//     Task_P2Main Outputs/GMotion.arrAxis[166].PlcToNc <-> Inputs/FromPlc
//   DPPLC/DPPLC Instance <-> NC-Task 1 SAF/Axes/Axis194_167 P3_M2_OvenRetracting
//     Task_P2Main Inputs/GMotion.arrAxis[167].NcToPlc <-> Outputs/ToPlc
//     Task_P2Main Outputs/GMotion.arrAxis[167].PlcToNc <-> Inputs/FromPlc
//   DPPLC/DPPLC Instance <-> NC-Task 1 SAF/Axes/Axis195_168 P3_M2_OvenUpDown
//     Task_P2Main Inputs/GMotion.arrAxis[168].NcToPlc <-> Outputs/ToPlc
//     Task_P2Main Outputs/GMotion.arrAxis[168].PlcToNc <-> Inputs/FromPlc
//   DPPLC/DPPLC Instance <-> NC-Task 1 SAF/Axes/Axis196_169 P3_M3_HotPressingLine
//     Task_P2Main Inputs/GMotion.arrAxis[169].NcToPlc <-> Outputs/ToPlc
//     Task_P2Main Outputs/GMotion.arrAxis[169].PlcToNc <-> Inputs/FromPlc
//   DPPLC/DPPLC Instance <-> NC-Task 1 SAF/Axes/Axis197_170 P3_M3_HotPressingActuated
//     Task_P2Main Inputs/GMotion.arrAxis[170].NcToPlc <-> Outputs/ToPlc
//     Task_P2Main Outputs/GMotion.arrAxis[170].PlcToNc <-> Inputs/FromPlc
//   DPPLC/DPPLC Instance <-> NC-Task 1 SAF/Axes/Axis198_171  P3_M4_WeighLine
//     Task_P2Main Inputs/GMotion.arrAxis[171].NcToPlc <-> Outputs/ToPlc
//     Task_P2Main Outputs/GMotion.arrAxis[171].PlcToNc <-> Inputs/FromPlc
//   DPPLC/DPPLC Instance <-> NC-Task 1 SAF/Axes/Axis199_172 P3_M4_WeighUpDown
//     Task_P2Main Inputs/GMotion.arrAxis[172].NcToPlc <-> Outputs/ToPlc
//     Task_P2Main Outputs/GMotion.arrAxis[172].PlcToNc <-> Inputs/FromPlc
//   DPPLC/DPPLC Instance <-> NC-Task 1 SAF/Axes/Axis200_173 P3_M4_WeighWhirling
//     Task_P2Main Inputs/GMotion.arrAxis[173].NcToPlc <-> Outputs/ToPlc
//     Task_P2Main Outputs/GMotion.arrAxis[173].PlcToNc <-> Inputs/FromPlc
//   DPPLC/DPPLC Instance <-> NC-Task 1 SAF/Axes/Axis201_174 P3_M4_SortingoutCarrying
//     Task_P2Main Inputs/GMotion.arrAxis[174].NcToPlc <-> Outputs/ToPlc
//     Task_P2Main Outputs/GMotion.arrAxis[174].PlcToNc <-> Inputs/FromPlc
//   DPPLC/DPPLC Instance <-> NC-Task 1 SAF/Axes/Axis202_175 P3_M4_SortingoutUpDown
//     Task_P2Main Inputs/GMotion.arrAxis[175].NcToPlc <-> Outputs/ToPlc
//     Task_P2Main Outputs/GMotion.arrAxis[175].PlcToNc <-> Inputs/FromPlc
//   DPPLC/DPPLC Instance <-> NC-Task 1 SAF/Axes/Axis203_176 P3_M4_OffloadingCarrying
//     Task_P2Main Inputs/GMotion.arrAxis[176].NcToPlc <-> Outputs/ToPlc
//     Task_P2Main Outputs/GMotion.arrAxis[176].PlcToNc <-> Inputs/FromPlc
//   DPPLC/DPPLC Instance <-> NC-Task 1 SAF/Axes/Axis204_177 P3_M4_OffloadingUpDown
//     Task_P2Main Inputs/GMotion.arrAxis[177].NcToPlc <-> Outputs/ToPlc
//     Task_P2Main Outputs/GMotion.arrAxis[177].PlcToNc <-> Inputs/FromPlc
//   DPPLC/DPPLC Instance <-> NC-Task 1 SAF/Axes/Axis205_178 P3_TapeAdvance
//     Task_P2Main Inputs/GMotion.arrAxis[178].NcToPlc <-> Outputs/ToPlc
//     Task_P2Main Outputs/GMotion.arrAxis[178].PlcToNc <-> Inputs/FromPlc
//   DPPLC/DPPLC Instance <-> NC-Task 1 SAF/Axes/Axis206_179 P3_TapeTranslation
//     Task_P2Main Inputs/GMotion.arrAxis[179].NcToPlc <-> Outputs/ToPlc
//     Task_P2Main Outputs/GMotion.arrAxis[179].PlcToNc <-> Inputs/FromPlc
//   DPPLC/DPPLC Instance <-> NC-Task 1 SAF/Axes/Axis207_180 P3_IDPut
//     Task_P2Main Inputs/GMotion.arrAxis[180].NcToPlc <-> Outputs/ToPlc
//     Task_P2Main Outputs/GMotion.arrAxis[180].PlcToNc <-> Inputs/FromPlc
//   DPPLC/DPPLC Instance <-> NC-Task 1 SAF/Axes/Axis208_181 P3_IDLift
//     Task_P2Main Inputs/GMotion.arrAxis[181].NcToPlc <-> Outputs/ToPlc
//     Task_P2Main Outputs/GMotion.arrAxis[181].PlcToNc <-> Inputs/FromPlc
//   DPPLC/DPPLC Instance <-> NC-Task 1 SAF/Axes/Axis209_182 P3_Standby5
//     Task_P2Main Inputs/GMotion.arrAxis[182].NcToPlc <-> Outputs/ToPlc
//     Task_P2Main Outputs/GMotion.arrAxis[182].PlcToNc <-> Inputs/FromPlc
//   DPPLC/DPPLC Instance <-> NC-Task 1 SAF/Axes/Axis218_153 P2M2_VirTimeWind
//     Task_P2Main Inputs/GMotion.arrAxis[153].NcToPlc <-> Outputs/ToPlc
//     Task_P2Main Outputs/GMotion.arrAxis[153].PlcToNc <-> Inputs/FromPlc
//   DPPLC/DPPLC Instance <-> NC-Task 1 SAF/Axes/Axis219_154 P2M3_VirTimeWind
//     Task_P2Main Inputs/GMotion.arrAxis[154].NcToPlc <-> Outputs/ToPlc
//     Task_P2Main Outputs/GMotion.arrAxis[154].PlcToNc <-> Inputs/FromPlc
//   DPPLC/DPPLC Instance <-> NC-Task 1 SAF/Axes/Axis220_140 P2M1_VirTimeWind
//     Task_P2Main Inputs/GMotion.arrAxis[140].NcToPlc <-> Outputs/ToPlc
//     Task_P2Main Outputs/GMotion.arrAxis[140].PlcToNc <-> Inputs/FromPlc
//   DPPLC/DPPLC Instance <-> NC-Task 1 SAF/Axes/Axis221_141 P2M1_VirMain
//     Task_P2Main Inputs/GMotion.arrAxis[141].NcToPlc <-> Outputs/ToPlc
//     Task_P2Main Outputs/GMotion.arrAxis[141].PlcToNc <-> Inputs/FromPlc
//   DPPLC/DPPLC Instance <-> NC-Task 1 SAF/Axes/Axis222_142 P2M1_VirDriver
//     Task_P2Main Inputs/GMotion.arrAxis[142].NcToPlc <-> Outputs/ToPlc
//     Task_P2Main Outputs/GMotion.arrAxis[142].PlcToNc <-> Inputs/FromPlc
//   DPPLC/DPPLC Instance <-> NC-Task 1 SAF/Axes/Axis223_143 P2M1_VirTailCurl
//     Task_P2Main Inputs/GMotion.arrAxis[143].NcToPlc <-> Outputs/ToPlc
//     Task_P2Main Outputs/GMotion.arrAxis[143].PlcToNc <-> Inputs/FromPlc
//   DPPLC/DPPLC Instance <-> NC-Task 1 SAF/Axes/Axis224_144  P2M1VirGM
//     Task_P2Main Inputs/GMotion.arrAxis[144].NcToPlc <-> Outputs/ToPlc
//     Task_P2Main Outputs/GMotion.arrAxis[144].PlcToNc <-> Inputs/FromPlc
//   DPPLC/DPPLC Instance <-> NC-Task 1 SAF/Axes/Axis225_145 P2M2_VirMain
//     Task_P2Main Inputs/GMotion.arrAxis[145].NcToPlc <-> Outputs/ToPlc
//     Task_P2Main Outputs/GMotion.arrAxis[145].PlcToNc <-> Inputs/FromPlc
//   DPPLC/DPPLC Instance <-> NC-Task 1 SAF/Axes/Axis226_146 P2M2_VirDriver
//     Task_P2Main Inputs/GMotion.arrAxis[146].NcToPlc <-> Outputs/ToPlc
//     Task_P2Main Outputs/GMotion.arrAxis[146].PlcToNc <-> Inputs/FromPlc
//   DPPLC/DPPLC Instance <-> NC-Task 1 SAF/Axes/Axis227_147 P2M2_VirTailCurl
//     Task_P2Main Inputs/GMotion.arrAxis[147].NcToPlc <-> Outputs/ToPlc
//     Task_P2Main Outputs/GMotion.arrAxis[147].PlcToNc <-> Inputs/FromPlc
//   DPPLC/DPPLC Instance <-> NC-Task 1 SAF/Axes/Axis228_148  P2M2VirGM
//     Task_P2Main Inputs/GMotion.arrAxis[148].NcToPlc <-> Outputs/ToPlc
//     Task_P2Main Outputs/GMotion.arrAxis[148].PlcToNc <-> Inputs/FromPlc
//   DPPLC/DPPLC Instance <-> NC-Task 1 SAF/Axes/Axis229_149 P2M3_VirMain
//     Task_P2Main Inputs/GMotion.arrAxis[149].NcToPlc <-> Outputs/ToPlc
//     Task_P2Main Outputs/GMotion.arrAxis[149].PlcToNc <-> Inputs/FromPlc
//   DPPLC/DPPLC Instance <-> NC-Task 1 SAF/Axes/Axis230_150 P2M3_VirDriver
//     Task_P2Main Inputs/GMotion.arrAxis[150].NcToPlc <-> Outputs/ToPlc
//     Task_P2Main Outputs/GMotion.arrAxis[150].PlcToNc <-> Inputs/FromPlc
//   DPPLC/DPPLC Instance <-> NC-Task 1 SAF/Axes/Axis231_151 P2M3_VirTailCurl
//     Task_P2Main Inputs/GMotion.arrAxis[151].NcToPlc <-> Outputs/ToPlc
//     Task_P2Main Outputs/GMotion.arrAxis[151].PlcToNc <-> Inputs/FromPlc
//   DPPLC/DPPLC Instance <-> NC-Task 1 SAF/Axes/Axis232  P2M3VirGM
//     Task_P2Main Inputs/GMotion.arrAxis[152].NcToPlc <-> Outputs/ToPlc
//     Task_P2Main Outputs/GMotion.arrAxis[152].PlcToNc <-> Inputs/FromPlc
//   DPPLC/DPPLC Instance <-> MQPLC/MQPLC Instance
//     Task_P2M3 Inputs/IO.M_Pro <-> Task_P1 Outputs/IO.M_Pro
//     Task_P2M3 Outputs/IO.D_Pro <-> Task_P1 Inputs/IO.D_Pro
//     Task_P2M3 Outputs/IO.D_Sys/P3ReadParDone <-> Task_P1 Inputs/IO.D_Sys/P3ReadParDone
//     Task_P2M3 Outputs/IO.D_Sys/P3SaveParDone <-> Task_P1 Inputs/IO.D_Sys/P3SaveParDone
//     Task_P2M3 Outputs/IO.D_Sys/bP2ClearDo <-> Task_P1 Inputs/IO.D_Sys/bP2ClearDo
//     Task_P2M3 Outputs/IO.D_Sys/bP2ClearDone <-> Task_P1 Inputs/IO.D_Sys/bP2ClearDone
//     Task_P2M3 Outputs/IO.D_Sys/bP2Estop <-> Task_P1 Inputs/IO.D_Sys/bP2Estop
//     Task_P2M3 Outputs/IO.D_Sys/bP2M1Enable <-> Task_P1 Inputs/IO.D_Sys/bP2M1Enable
//     Task_P2M3 Outputs/IO.D_Sys/bP2M2Enable <-> Task_P1 Inputs/IO.D_Sys/bP2M2Enable
//     Task_P2M3 Outputs/IO.D_Sys/bP2M3Enable <-> Task_P1 Inputs/IO.D_Sys/bP2M3Enable
//     Task_P2M3 Outputs/IO.D_Sys/bP2Runing <-> Task_P1 Inputs/IO.D_Sys/bP2Runing
//     Task_P2M3 Outputs/IO.D_Sys/bP2Start <-> Task_P1 Inputs/IO.D_Sys/bP2Start
//     Task_P2M3 Outputs/IO.D_Sys/fM1MainSetPos <-> Task_P1 Inputs/IO.D_Sys/fM1MainSetPos
//     Task_P2M3 Outputs/IO.D_Sys/fM2MainSetPos <-> Task_P1 Inputs/IO.D_Sys/fM2MainSetPos
//     Task_P2M3 Outputs/IO.D_Sys/fM3MainSetPos <-> Task_P1 Inputs/IO.D_Sys/fM3MainSetPos
//     Task_P2M3 Outputs/IO.D_Sys/iAn1Ask <-> Task_P1 Inputs/IO.D_Sys/iAn1Ask
//     Task_P2M3 Outputs/IO.D_Sys/iAn2Ask <-> Task_P1 Inputs/IO.D_Sys/iAn2Ask
//     Task_P2M3 Outputs/IO.D_Sys/iAn3Ask <-> Task_P1 Inputs/IO.D_Sys/iAn3Ask
//     Task_P2M3 Outputs/IO.D_Sys/iCa1Ask <-> Task_P1 Inputs/IO.D_Sys/iCa1Ask
//     Task_P2M3 Outputs/IO.D_Sys/iCa2Ask <-> Task_P1 Inputs/IO.D_Sys/iCa2Ask
//     Task_P2M3 Outputs/IO.D_Sys/iCa3Ask <-> Task_P1 Inputs/IO.D_Sys/iCa3Ask
//     Task_P2Main Inputs/IO.AnMQ_MES1 <-> Task_P1 Outputs/IO.AnMQ_MES1
//     Task_P2Main Inputs/IO.AnMQ_MES2 <-> Task_P1 Outputs/IO.AnMQ_MES2
//     Task_P2Main Inputs/IO.AnMQ_MES3 <-> Task_P1 Outputs/IO.AnMQ_MES3
//     Task_P2Main Inputs/IO.CaMQ_MES1 <-> Task_P1 Outputs/IO.CaMQ_MES1
//     Task_P2Main Inputs/IO.CaMQ_MES2 <-> Task_P1 Outputs/IO.CaMQ_MES2
//     Task_P2Main Inputs/IO.CaMQ_MES3 <-> Task_P1 Outputs/IO.CaMQ_MES3
//     Task_P2Main Outputs/IO.YL_Q <-> Task_P1 Inputs/IO.YL_I
//     Task_P3 Inputs/IO.M_Sys/P1ReadParDone <-> Task_P1 Outputs/IO.M_Sys/P1ReadParDone
//     Task_P3 Inputs/IO.M_Sys/P1SaveParDone <-> Task_P1 Outputs/IO.M_Sys/P1SaveParDone
//     Task_P3 Inputs/IO.M_Sys/bP1ClearDo <-> Task_P1 Outputs/IO.M_Sys/bP1ClearDo
//     Task_P3 Inputs/IO.M_Sys/bP1ClearDone <-> Task_P1 Outputs/IO.M_Sys/bP1ClearDone
//     Task_P3 Inputs/IO.M_Sys/bP1Estop <-> Task_P1 Outputs/IO.M_Sys/bP1Estop
//     Task_P3 Inputs/IO.M_Sys/bP1Runing <-> Task_P1 Outputs/IO.M_Sys/bP1Runing
//     Task_P3 Inputs/IO.M_Sys/bP1Start <-> Task_P1 Outputs/IO.M_Sys/bP1Start
//     Task_P3 Inputs/IO.M_Sys/iCarryPoleMode <-> Task_P1 Outputs/IO.M_Sys/iCarryPoleMode
//     Task_P3 Inputs/IO.M_Sys/p1state <-> Task_P1 Outputs/IO.M_Sys/p1state
//     Task_P3 Inputs/IO.YL_INT1 <-> Task_P1 Outputs/IO.YL_INT1
//     Task_P3 Inputs/P3IO.MTD_Mes1/bFuncEN <-> Task_P1 Outputs/IO.MTD_Mes1/bFuncEN
//     Task_P3 Inputs/P3IO.MTD_Mes1/rExcelRate <-> Task_P1 Outputs/IO.MTD_Mes1/rExcelRate
//     Task_P3 Inputs/P3IO.MTD_Mes1/uOther <-> Task_P1 Outputs/IO.MTD_Mes1/uOther
//     Task_P3 Inputs/P3Par.MQ_To_DT_MES <-> Task_P1 Outputs/IO.MQ_To_DT_MES
//     Task_P3 Outputs/IO.YL_INT2 <-> Task_P1 Inputs/IO.YL_INT2
//     Task_P3 Outputs/P3IO.DTM_Mes1/bFuncEN <-> Task_P1 Inputs/IO.DTM_Mes1/bFuncEN
//     Task_P3 Outputs/P3IO.DTM_Mes1/uOther <-> Task_P1 Inputs/IO.DTM_Mes1/uOther
//     Task_P3 Outputs/P3Par.DT_To_MQ_MES <-> Task_P1 Inputs/IO.DT_To_MQ_MES
//   MQPLC/MQPLC Instance <-> Device 3 (EtherCAT)/Box 2 (CU1128)/Term 24 (CU1128-B)/负极上表面除尘皮带(InoSV660N)
//     Task_P1 Inputs/GMotion.DrivesOP[42] <-> InfoData/State
//     Task_P1 Inputs/GMotion.arrAxisCtrl[42].Io.DigitalInputs <-> Inputs/Digital inputs
//     Task_P1 Inputs/GMotion.arrAxisCtrl[42].Io.ErrorCode <-> Inputs/Error code
//     Task_P1 Inputs/GMotion.iActTorque_M[42] <-> Inputs/Torque actual value
//   MQPLC/MQPLC Instance <-> Device 3 (EtherCAT)/Box 2 (CU1128)/Term 24 (CU1128-B)/负极下表面除尘倒装皮带(InoSV660N)
//     Task_P1 Inputs/GMotion.DrivesOP[43] <-> InfoData/State
//     Task_P1 Inputs/GMotion.arrAxisCtrl[43].Io.DigitalInputs <-> Inputs/Digital inputs
//     Task_P1 Inputs/GMotion.arrAxisCtrl[43].Io.ErrorCode <-> Inputs/Error code
//     Task_P1 Inputs/GMotion.iActTorque_M[43] <-> Inputs/Torque actual value
//   MQPLC/MQPLC Instance <-> Device 3 (EtherCAT)/Box 2 (CU1128)/Term 24 (CU1128-B)/负极倒角模具(InoSV660N)
//     Task_P1 Inputs/GMotion.DrivesOP[30] <-> InfoData/State
//     Task_P1 Inputs/GMotion.arrAxisCtrl[30].Io.DigitalInputs <-> Inputs/Digital inputs
//     Task_P1 Inputs/GMotion.arrAxisCtrl[30].Io.ErrorCode <-> Inputs/Error code
//     Task_P1 Inputs/GMotion.iActTorque_M[30] <-> Inputs/Torque actual value
//   MQPLC/MQPLC Instance <-> Device 3 (EtherCAT)/Box 2 (CU1128)/Term 24 (CU1128-B)/负极右放卷电机(InoSV660N)
//     Task_P1 Inputs/GMotion.DrivesOP[26] <-> InfoData/State
//     Task_P1 Inputs/GMotion.arrAxisCtrl[26].Io.DigitalInputs <-> Inputs/Digital inputs
//     Task_P1 Inputs/GMotion.arrAxisCtrl[26].Io.ErrorCode <-> Inputs/Error code
//     Task_P1 Inputs/GMotion.iActTorque_M[26] <-> Inputs/Torque actual value
//   MQPLC/MQPLC Instance <-> Device 3 (EtherCAT)/Box 2 (CU1128)/Term 24 (CU1128-B)/负极尺寸CCD压片升降(InoSV660N)
//     Task_P1 Inputs/GMotion.DrivesOP[38] <-> InfoData/State
//     Task_P1 Inputs/GMotion.arrAxisCtrl[38].Io.DigitalInputs <-> Inputs/Digital inputs
//     Task_P1 Inputs/GMotion.arrAxisCtrl[38].Io.ErrorCode <-> Inputs/Error code
//     Task_P1 Inputs/GMotion.iActTorque_M[38] <-> Inputs/Torque actual value
//   MQPLC/MQPLC Instance <-> Device 3 (EtherCAT)/Box 2 (CU1128)/Term 24 (CU1128-B)/负极左放卷电机(InoSV660N)
//     Task_P1 Inputs/GMotion.DrivesOP[25] <-> InfoData/State
//     Task_P1 Inputs/GMotion.arrAxisCtrl[25].Io.DigitalInputs <-> Inputs/Digital inputs
//     Task_P1 Inputs/GMotion.arrAxisCtrl[25].Io.ErrorCode <-> Inputs/Error code
//     Task_P1 Inputs/GMotion.iActTorque_M[25] <-> Inputs/Torque actual value
//   MQPLC/MQPLC Instance <-> Device 3 (EtherCAT)/Box 2 (CU1128)/Term 24 (CU1128-B)/负极模具纠偏X轴(肩宽)(InoSV660N)
//     Task_P1 Inputs/GMotion.DrivesOP[31] <-> InfoData/State
//     Task_P1 Inputs/GMotion.arrAxisCtrl[31].Io.DigitalInputs <-> Inputs/Digital inputs
//     Task_P1 Inputs/GMotion.arrAxisCtrl[31].Io.ErrorCode <-> Inputs/Error code
//     Task_P1 Inputs/GMotion.iActTorque_M[31] <-> Inputs/Torque actual value
//   MQPLC/MQPLC Instance <-> Device 3 (EtherCAT)/Box 2 (CU1128)/Term 24 (CU1128-B)/负极模具纠偏Y轴(InoSV660N)
//     Task_P1 Inputs/GMotion.DrivesOP[32] <-> InfoData/State
//     Task_P1 Inputs/GMotion.arrAxisCtrl[32].Io.DigitalInputs <-> Inputs/Digital inputs
//     Task_P1 Inputs/GMotion.arrAxisCtrl[32].Io.ErrorCode <-> Inputs/Error code
//     Task_P1 Inputs/GMotion.iActTorque_M[32] <-> Inputs/Torque actual value
//   MQPLC/MQPLC Instance <-> Device 3 (EtherCAT)/Box 2 (CU1128)/Term 24 (CU1128-B)/负极模切主驱动(CDHD)
//     Task_P1 Inputs/GMotion.DrivesOP[33] <-> InfoData/State
//     Task_P1 Inputs/GMotion.arrAxisCtrl[33].Io.DigitalInputs <-> TxPDO 4/Digital inputs
//     Task_P1 Inputs/GMotion.iActTorque_M[33] <-> TxPDO 1/Torque Actual Value
//   MQPLC/MQPLC Instance <-> Device 3 (EtherCAT)/Box 2 (CU1128)/Term 24 (CU1128-B)/负极模切前摆杆张力(InoSV660N)
//     Task_P1 Inputs/GMotion.DrivesOP[27] <-> InfoData/State
//     Task_P1 Inputs/GMotion.arrAxisCtrl[27].Io.DigitalInputs <-> Inputs/Digital inputs
//     Task_P1 Inputs/GMotion.arrAxisCtrl[27].Io.ErrorCode <-> Inputs/Error code
//     Task_P1 Inputs/GMotion.iActDriveTorque[2] <-> Inputs/Torque actual value
//     Task_P1 Outputs/GMotion.iMaxProfileVelo[2] <-> Outputs/Max profile velocity
//     Task_P1 Outputs/GMotion.iNegtiveTorqueLimits[2] <-> Outputs/Negative torque limit value
//     Task_P1 Outputs/GMotion.iPostiveTorqueLimits[2] <-> Outputs/Positive torque limit value
//     Task_P1 Outputs/GMotion.iSetDriveMode[2] <-> Outputs/Modes of operation
//     Task_P1 Outputs/GMotion.iTargetTorque[2] <-> Outputs/Target torque
//   MQPLC/MQPLC Instance <-> Device 3 (EtherCAT)/Box 2 (CU1128)/Term 24 (CU1128-B)/负极模切极片缓存(CDHD)
//     Task_P1 Inputs/GMotion.DrivesOP[29] <-> InfoData/State
//     Task_P1 Inputs/GMotion.arrAxisCtrl[29].Io.DigitalInputs <-> TxPDO 4/Digital inputs
//     Task_P1 Inputs/GMotion.iActTorque_M[29] <-> TxPDO 1/Torque Actual Value
//   MQPLC/MQPLC Instance <-> Device 3 (EtherCAT)/Box 2 (CU1128)/Term 24 (CU1128-B)/负极模切辅助驱动(InoSV660N)
//     Task_P1 Inputs/GMotion.DrivesOP[28] <-> InfoData/State
//     Task_P1 Inputs/GMotion.arrAxisCtrl[28].Io.DigitalInputs <-> Inputs/Digital inputs
//     Task_P1 Inputs/GMotion.arrAxisCtrl[28].Io.ErrorCode <-> Inputs/Error code
//     Task_P1 Inputs/GMotion.iActTorque_M[28] <-> Inputs/Torque actual value
//   MQPLC/MQPLC Instance <-> Device 3 (EtherCAT)/Box 2 (CU1128)/Term 24 (CU1128-B)/负极裁切切刀(InoSV660N)
//     Task_P1 Inputs/GMotion.DrivesOP[34] <-> InfoData/State
//     Task_P1 Inputs/GMotion.arrAxisCtrl[34].Io.DigitalInputs <-> Inputs/Digital inputs
//     Task_P1 Inputs/GMotion.arrAxisCtrl[34].Io.ErrorCode <-> Inputs/Error code
//     Task_P1 Inputs/GMotion.iActTorque_M[34] <-> Inputs/Torque actual value
//   MQPLC/MQPLC Instance <-> Device 3 (EtherCAT)/Box 2 (CU1128)/Term 24 (CU1128-B)/负极裁切角度纠偏(InoSV660N)
//     Task_P1 Inputs/GMotion.DrivesOP[35] <-> InfoData/State
//     Task_P1 Inputs/GMotion.arrAxisCtrl[35].Io.DigitalInputs <-> Inputs/Digital inputs
//     Task_P1 Inputs/GMotion.arrAxisCtrl[35].Io.ErrorCode <-> Inputs/Error code
//     Task_P1 Inputs/GMotion.iActTorque_M[35] <-> Inputs/Torque actual value
//   MQPLC/MQPLC Instance <-> Device 3 (EtherCAT)/Box 2 (CU1128)/Term 24 (CU1128-B)/负极裁切输送带换型(InoSV660N)
//     Task_P1 Inputs/GMotion.DrivesOP[37] <-> InfoData/State
//     Task_P1 Inputs/GMotion.arrAxisCtrl[37].Io.DigitalInputs <-> Inputs/Digital inputs
//     Task_P1 Inputs/GMotion.arrAxisCtrl[37].Io.ErrorCode <-> Inputs/Error code
//     Task_P1 Inputs/GMotion.iActTorque_M[37] <-> Inputs/Torque actual value
//   MQPLC/MQPLC Instance <-> Device 3 (EtherCAT)/Box 2 (CU1128)/Term 24 (CU1128-B)/负极裁切输送皮带(InoSV660N)
//     Task_P1 Inputs/GMotion.DrivesOP[36] <-> InfoData/State
//     Task_P1 Inputs/GMotion.arrAxisCtrl[36].Io.DigitalInputs <-> Inputs/Digital inputs
//     Task_P1 Inputs/GMotion.arrAxisCtrl[36].Io.ErrorCode <-> Inputs/Error code
//     Task_P1 Inputs/GMotion.iActTorque_M[36] <-> Inputs/Torque actual value
//   MQPLC/MQPLC Instance <-> Device 3 (EtherCAT)/Box 2 (CU1128)/Term 24 (CU1128-B)/负极踢单张废料(InoSV660N)
//     Task_P1 Inputs/GMotion.DrivesOP[41] <-> InfoData/State
//     Task_P1 Inputs/GMotion.arrAxisCtrl[41].Io.DigitalInputs <-> Inputs/Digital inputs
//     Task_P1 Inputs/GMotion.arrAxisCtrl[41].Io.ErrorCode <-> Inputs/Error code
//     Task_P1 Inputs/GMotion.iActTorque_M[41] <-> Inputs/Torque actual value
//   MQPLC/MQPLC Instance <-> Device 3 (EtherCAT)/Box 2 (CU1128)/Term 24 (CU1128-B)/负极踢废倒装皮带(InoSV660N)
//     Task_P1 Inputs/GMotion.DrivesOP[39] <-> InfoData/State
//     Task_P1 Inputs/GMotion.arrAxisCtrl[39].Io.DigitalInputs <-> Inputs/Digital inputs
//     Task_P1 Inputs/GMotion.arrAxisCtrl[39].Io.ErrorCode <-> Inputs/Error code
//     Task_P1 Inputs/GMotion.iActTorque_M[39] <-> Inputs/Torque actual value
//   MQPLC/MQPLC Instance <-> Device 3 (EtherCAT)/Box 2 (CU1128)/Term 24 (CU1128-B)/负极踢连续废料(InoSV660N)
//     Task_P1 Inputs/GMotion.DrivesOP[40] <-> InfoData/State
//     Task_P1 Inputs/GMotion.arrAxisCtrl[40].Io.DigitalInputs <-> Inputs/Digital inputs
//     Task_P1 Inputs/GMotion.arrAxisCtrl[40].Io.ErrorCode <-> Inputs/Error code
//     Task_P1 Inputs/GMotion.iActTorque_M[40] <-> Inputs/Torque actual value
//   MQPLC/MQPLC Instance <-> Device 3 (EtherCAT)/Box 2 (CU1128)/Term 44 (CU1128-C)/P2M2正极送料分段皮带2[21(模切)] (InoSV660N)
//     Task_P1 Inputs/GMotion.arrAxisCtrl[21].Io.ErrorCode <-> Inputs/Error code
//     Task_P1 Inputs/GMotion.iActTorque_M[21] <-> Inputs/Torque actual value
//   MQPLC/MQPLC Instance <-> Device 3 (EtherCAT)/Box 2 (CU1128)/Term 44 (CU1128-C)/P2M2负极送料分段皮带2（45模切） (InoSV660N)
//     Task_P1 Inputs/GMotion.arrAxisCtrl[45].Io.ErrorCode <-> Inputs/Error code
//     Task_P1 Inputs/GMotion.iActTorque_M[45] <-> Inputs/Torque actual value
//   MQPLC/MQPLC Instance <-> Device 3 (EtherCAT)/Box 2 (CU1128)/Term 44 (CU1128-C)/P2M3正极送料分段皮带3（22模切） (InoSV660N)
//     Task_P1 Inputs/GMotion.arrAxisCtrl[22].Io.ErrorCode <-> Inputs/Error code
//     Task_P1 Inputs/GMotion.iActTorque_M[22] <-> Inputs/Torque actual value
//   MQPLC/MQPLC Instance <-> Device 3 (EtherCAT)/Box 2 (CU1128)/Term 44 (CU1128-C)/P2M3负极送料分段皮带3（46模切） (InoSV660N)
//     Task_P1 Inputs/GMotion.arrAxisCtrl[46].Io.ErrorCode <-> Inputs/Error code
//     Task_P1 Inputs/GMotion.iActTorque_M[46] <-> Inputs/Torque actual value
//   MQPLC/MQPLC Instance <-> Device 3 (EtherCAT)/Box 2 (CU1128)/一号叠片IO耦合器(GSIO-A-ECC)
//     Task_P1 Inputs/IO.I30101 <-> I301/Digital Inputs/Channel 1
//     Task_P1 Inputs/IO.I30107 <-> I301/Digital Inputs/Channel 7
//     Task_P1 Outputs/IO.Q30103 <-> Q301/Digital Outputs/Channel 3
//     Task_P1 Outputs/IO.Q30104 <-> Q301/Digital Outputs/Channel 4
//     Task_P1 Outputs/IO.Q30201 <-> Q302/Digital Outputs/Channel 1
//     Task_P1 Outputs/IO.Q30202 <-> Q302/Digital Outputs/Channel 2
//   MQPLC/MQPLC Instance <-> Device 3 (EtherCAT)/Box 2 (CU1128)/三号叠片IO耦合器(GSIO-A-ECC)
//     Task_P1 Inputs/IO.I50101 <-> I501 (GSIO-A-16DIN)/Digital Inputs/Channel 1
//     Task_P1 Inputs/IO.I50107 <-> I501 (GSIO-A-16DIN)/Digital Inputs/Channel 7
//     Task_P1 Outputs/IO.Q50103 <-> Q501 (GSIO-A-16DON)/Digital Outputs/Channel 3
//     Task_P1 Outputs/IO.Q50104 <-> Q501 (GSIO-A-16DON)/Digital Outputs/Channel 4
//     Task_P1 Outputs/IO.Q50201 <-> Q502 (GSIO-A-16DON)/Digital Outputs/Channel 1
//     Task_P1 Outputs/IO.Q50202 <-> Q502 (GSIO-A-16DON)/Digital Outputs/Channel 2
//   MQPLC/MQPLC Instance <-> Device 3 (EtherCAT)/Box 2 (CU1128)/二号叠片IO耦合器 (GSIO-A-ECC)
//     Task_P1 Inputs/IO.I40101 <-> I401 (GSIO-A-16DIN)/Digital Inputs/Channel 1
//     Task_P1 Inputs/IO.I40107 <-> I401 (GSIO-A-16DIN)/Digital Inputs/Channel 7
//     Task_P1 Outputs/IO.Q40103 <-> O401 (GSIO-A-16DON)/Digital Outputs/Channel 3
//     Task_P1 Outputs/IO.Q40104 <-> O401 (GSIO-A-16DON)/Digital Outputs/Channel 4
//     Task_P1 Outputs/IO.Q40201 <-> O402 (GSIO-A-16DON)/Digital Outputs/Channel 1
//     Task_P1 Outputs/IO.Q40202 <-> O402 (GSIO-A-16DON)/Digital Outputs/Channel 2
//   MQPLC/MQPLC Instance <-> Device 3 (EtherCAT)/Box 2 (CU1128)/正极IO耦合器(GSIO-A-ECC)
//     Task_P1 Inputs/IO.AI101[0] <-> AI101 (GSIO-A-4AIHV)/Analog Inputs/Channel 1
//     Task_P1 Inputs/IO.AI101[1] <-> AI101 (GSIO-A-4AIHV)/Analog Inputs/Channel 2
//     Task_P1 Inputs/IO.AI101[2] <-> AI101 (GSIO-A-4AIHV)/Analog Inputs/Channel 3
//     Task_P1 Inputs/IO.AI101[3] <-> AI101 (GSIO-A-4AIHV)/Analog Inputs/Channel 4
//     Task_P1 Inputs/IO.AI102[0] <-> AI102 (GSIO-A-4AIHV)/Analog Inputs/Channel 1
//     Task_P1 Inputs/IO.AI102[1] <-> AI102 (GSIO-A-4AIHV)/Analog Inputs/Channel 2
//     Task_P1 Inputs/IO.AI102[2] <-> AI102 (GSIO-A-4AIHV)/Analog Inputs/Channel 3
//     Task_P1 Inputs/IO.AI102[3] <-> AI102 (GSIO-A-4AIHV)/Analog Inputs/Channel 4
//     Task_P1 Inputs/IO.I101[10] <-> I101 (GSIO-A-16DIN)/Digital Inputs/Channel 10
//     Task_P1 Inputs/IO.I101[11] <-> I101 (GSIO-A-16DIN)/Digital Inputs/Channel 11
//     Task_P1 Inputs/IO.I101[12] <-> I101 (GSIO-A-16DIN)/Digital Inputs/Channel 12
//     Task_P1 Inputs/IO.I101[13] <-> I101 (GSIO-A-16DIN)/Digital Inputs/Channel 13
//     Task_P1 Inputs/IO.I101[14] <-> I101 (GSIO-A-16DIN)/Digital Inputs/Channel 14
//     Task_P1 Inputs/IO.I101[15] <-> I101 (GSIO-A-16DIN)/Digital Inputs/Channel 15
//     Task_P1 Inputs/IO.I101[16] <-> I101 (GSIO-A-16DIN)/Digital Inputs/Channel 16
//     Task_P1 Inputs/IO.I101[1] <-> I101 (GSIO-A-16DIN)/Digital Inputs/Channel 1
//     Task_P1 Inputs/IO.I101[2] <-> I101 (GSIO-A-16DIN)/Digital Inputs/Channel 2
//     Task_P1 Inputs/IO.I101[3] <-> I101 (GSIO-A-16DIN)/Digital Inputs/Channel 3
//     Task_P1 Inputs/IO.I101[4] <-> I101 (GSIO-A-16DIN)/Digital Inputs/Channel 4
//     Task_P1 Inputs/IO.I101[5] <-> I101 (GSIO-A-16DIN)/Digital Inputs/Channel 5
//     Task_P1 Inputs/IO.I101[6] <-> I101 (GSIO-A-16DIN)/Digital Inputs/Channel 6
//     Task_P1 Inputs/IO.I101[7] <-> I101 (GSIO-A-16DIN)/Digital Inputs/Channel 7
//     Task_P1 Inputs/IO.I101[8] <-> I101 (GSIO-A-16DIN)/Digital Inputs/Channel 8
//     Task_P1 Inputs/IO.I101[9] <-> I101 (GSIO-A-16DIN)/Digital Inputs/Channel 9
//     Task_P1 Inputs/IO.I102[10] <-> I102 (GSIO-A-16DIN)/Digital Inputs/Channel 10
//     Task_P1 Inputs/IO.I102[11] <-> I102 (GSIO-A-16DIN)/Digital Inputs/Channel 11
//     Task_P1 Inputs/IO.I102[12] <-> I102 (GSIO-A-16DIN)/Digital Inputs/Channel 12
//     Task_P1 Inputs/IO.I102[13] <-> I102 (GSIO-A-16DIN)/Digital Inputs/Channel 13
//     Task_P1 Inputs/IO.I102[14] <-> I102 (GSIO-A-16DIN)/Digital Inputs/Channel 14
//     Task_P1 Inputs/IO.I102[15] <-> I102 (GSIO-A-16DIN)/Digital Inputs/Channel 15
//     Task_P1 Inputs/IO.I102[16] <-> I102 (GSIO-A-16DIN)/Digital Inputs/Channel 16
//     Task_P1 Inputs/IO.I102[1] <-> I102 (GSIO-A-16DIN)/Digital Inputs/Channel 1
//     Task_P1 Inputs/IO.I102[2] <-> I102 (GSIO-A-16DIN)/Digital Inputs/Channel 2
//     Task_P1 Inputs/IO.I102[3] <-> I102 (GSIO-A-16DIN)/Digital Inputs/Channel 3
//     Task_P1 Inputs/IO.I102[4] <-> I102 (GSIO-A-16DIN)/Digital Inputs/Channel 4
//     Task_P1 Inputs/IO.I102[5] <-> I102 (GSIO-A-16DIN)/Digital Inputs/Channel 5
//     Task_P1 Inputs/IO.I102[6] <-> I102 (GSIO-A-16DIN)/Digital Inputs/Channel 6
//     Task_P1 Inputs/IO.I102[7] <-> I102 (GSIO-A-16DIN)/Digital Inputs/Channel 7
//     Task_P1 Inputs/IO.I102[8] <-> I102 (GSIO-A-16DIN)/Digital Inputs/Channel 8
//     Task_P1 Inputs/IO.I102[9] <-> I102 (GSIO-A-16DIN)/Digital Inputs/Channel 9
//     Task_P1 Inputs/IO.I103[10] <-> I103 (GSIO-A-16DIN)/Digital Inputs/Channel 10
//     Task_P1 Inputs/IO.I103[11] <-> I103 (GSIO-A-16DIN)/Digital Inputs/Channel 11
//     Task_P1 Inputs/IO.I103[12] <-> I103 (GSIO-A-16DIN)/Digital Inputs/Channel 12
//     Task_P1 Inputs/IO.I103[13] <-> I103 (GSIO-A-16DIN)/Digital Inputs/Channel 13
//     Task_P1 Inputs/IO.I103[14] <-> I103 (GSIO-A-16DIN)/Digital Inputs/Channel 14
//     Task_P1 Inputs/IO.I103[15] <-> I103 (GSIO-A-16DIN)/Digital Inputs/Channel 15
//     Task_P1 Inputs/IO.I103[16] <-> I103 (GSIO-A-16DIN)/Digital Inputs/Channel 16
//     Task_P1 Inputs/IO.I103[1] <-> I103 (GSIO-A-16DIN)/Digital Inputs/Channel 1
//     Task_P1 Inputs/IO.I103[2] <-> I103 (GSIO-A-16DIN)/Digital Inputs/Channel 2
//     Task_P1 Inputs/IO.I103[3] <-> I103 (GSIO-A-16DIN)/Digital Inputs/Channel 3
//     Task_P1 Inputs/IO.I103[4] <-> I103 (GSIO-A-16DIN)/Digital Inputs/Channel 4
//     Task_P1 Inputs/IO.I103[5] <-> I103 (GSIO-A-16DIN)/Digital Inputs/Channel 5
//     Task_P1 Inputs/IO.I103[6] <-> I103 (GSIO-A-16DIN)/Digital Inputs/Channel 6
//     Task_P1 Inputs/IO.I103[7] <-> I103 (GSIO-A-16DIN)/Digital Inputs/Channel 7
//     Task_P1 Inputs/IO.I103[8] <-> I103 (GSIO-A-16DIN)/Digital Inputs/Channel 8
//     Task_P1 Inputs/IO.I103[9] <-> I103 (GSIO-A-16DIN)/Digital Inputs/Channel 9
//     Task_P1 Inputs/IO.I104[10] <-> I104 (GSIO-A-16DIN)/Digital Inputs/Channel 10
//     Task_P1 Inputs/IO.I104[11] <-> I104 (GSIO-A-16DIN)/Digital Inputs/Channel 11
//     Task_P1 Inputs/IO.I104[12] <-> I104 (GSIO-A-16DIN)/Digital Inputs/Channel 12
//     Task_P1 Inputs/IO.I104[13] <-> I104 (GSIO-A-16DIN)/Digital Inputs/Channel 13
//     Task_P1 Inputs/IO.I104[14] <-> I104 (GSIO-A-16DIN)/Digital Inputs/Channel 14
//     Task_P1 Inputs/IO.I104[15] <-> I104 (GSIO-A-16DIN)/Digital Inputs/Channel 15
//     Task_P1 Inputs/IO.I104[16] <-> I104 (GSIO-A-16DIN)/Digital Inputs/Channel 16
//     Task_P1 Inputs/IO.I104[1] <-> I104 (GSIO-A-16DIN)/Digital Inputs/Channel 1
//     Task_P1 Inputs/IO.I104[2] <-> I104 (GSIO-A-16DIN)/Digital Inputs/Channel 2
//     Task_P1 Inputs/IO.I104[3] <-> I104 (GSIO-A-16DIN)/Digital Inputs/Channel 3
//     Task_P1 Inputs/IO.I104[4] <-> I104 (GSIO-A-16DIN)/Digital Inputs/Channel 4
//     Task_P1 Inputs/IO.I104[5] <-> I104 (GSIO-A-16DIN)/Digital Inputs/Channel 5
//     Task_P1 Inputs/IO.I104[6] <-> I104 (GSIO-A-16DIN)/Digital Inputs/Channel 6
//     Task_P1 Inputs/IO.I104[7] <-> I104 (GSIO-A-16DIN)/Digital Inputs/Channel 7
//     Task_P1 Inputs/IO.I104[8] <-> I104 (GSIO-A-16DIN)/Digital Inputs/Channel 8
//     Task_P1 Inputs/IO.I104[9] <-> I104 (GSIO-A-16DIN)/Digital Inputs/Channel 9
//     Task_P1 Inputs/IO.I105[10] <-> I105 (GSIO-A-16DIN)/Digital Inputs/Channel 10
//     Task_P1 Inputs/IO.I105[11] <-> I105 (GSIO-A-16DIN)/Digital Inputs/Channel 11
//     Task_P1 Inputs/IO.I105[12] <-> I105 (GSIO-A-16DIN)/Digital Inputs/Channel 12
//     Task_P1 Inputs/IO.I105[13] <-> I105 (GSIO-A-16DIN)/Digital Inputs/Channel 13
//     Task_P1 Inputs/IO.I105[14] <-> I105 (GSIO-A-16DIN)/Digital Inputs/Channel 14
//     Task_P1 Inputs/IO.I105[15] <-> I105 (GSIO-A-16DIN)/Digital Inputs/Channel 15
//     Task_P1 Inputs/IO.I105[16] <-> I105 (GSIO-A-16DIN)/Digital Inputs/Channel 16
//     Task_P1 Inputs/IO.I105[1] <-> I105 (GSIO-A-16DIN)/Digital Inputs/Channel 1
//     Task_P1 Inputs/IO.I105[2] <-> I105 (GSIO-A-16DIN)/Digital Inputs/Channel 2
//     Task_P1 Inputs/IO.I105[3] <-> I105 (GSIO-A-16DIN)/Digital Inputs/Channel 3
//     Task_P1 Inputs/IO.I105[4] <-> I105 (GSIO-A-16DIN)/Digital Inputs/Channel 4
//     Task_P1 Inputs/IO.I105[5] <-> I105 (GSIO-A-16DIN)/Digital Inputs/Channel 5
//     Task_P1 Inputs/IO.I105[6] <-> I105 (GSIO-A-16DIN)/Digital Inputs/Channel 6
//     Task_P1 Inputs/IO.I105[7] <-> I105 (GSIO-A-16DIN)/Digital Inputs/Channel 7
//     Task_P1 Inputs/IO.I105[8] <-> I105 (GSIO-A-16DIN)/Digital Inputs/Channel 8
//     Task_P1 Inputs/IO.I105[9] <-> I105 (GSIO-A-16DIN)/Digital Inputs/Channel 9
//     Task_P1 Inputs/IO.I106[10] <-> I106 (GSIO-A-16DIN)/Digital Inputs/Channel 10
//     Task_P1 Inputs/IO.I106[11] <-> I106 (GSIO-A-16DIN)/Digital Inputs/Channel 11
//     Task_P1 Inputs/IO.I106[12] <-> I106 (GSIO-A-16DIN)/Digital Inputs/Channel 12
//     Task_P1 Inputs/IO.I106[13] <-> I106 (GSIO-A-16DIN)/Digital Inputs/Channel 13
//     Task_P1 Inputs/IO.I106[14] <-> I106 (GSIO-A-16DIN)/Digital Inputs/Channel 14
//     Task_P1 Inputs/IO.I106[15] <-> I106 (GSIO-A-16DIN)/Digital Inputs/Channel 15
//     Task_P1 Inputs/IO.I106[16] <-> I106 (GSIO-A-16DIN)/Digital Inputs/Channel 16
//     Task_P1 Inputs/IO.I106[1] <-> I106 (GSIO-A-16DIN)/Digital Inputs/Channel 1
//     Task_P1 Inputs/IO.I106[2] <-> I106 (GSIO-A-16DIN)/Digital Inputs/Channel 2
//     Task_P1 Inputs/IO.I106[3] <-> I106 (GSIO-A-16DIN)/Digital Inputs/Channel 3
//     Task_P1 Inputs/IO.I106[4] <-> I106 (GSIO-A-16DIN)/Digital Inputs/Channel 4
//     Task_P1 Inputs/IO.I106[5] <-> I106 (GSIO-A-16DIN)/Digital Inputs/Channel 5
//     Task_P1 Inputs/IO.I106[6] <-> I106 (GSIO-A-16DIN)/Digital Inputs/Channel 6
//     Task_P1 Inputs/IO.I106[7] <-> I106 (GSIO-A-16DIN)/Digital Inputs/Channel 7
//     Task_P1 Inputs/IO.I106[8] <-> I106 (GSIO-A-16DIN)/Digital Inputs/Channel 8
//     Task_P1 Inputs/IO.I106[9] <-> I106 (GSIO-A-16DIN)/Digital Inputs/Channel 9
//     Task_P1 Inputs/IO.I107[10] <-> I107 (GSIO-A-16DIN)/Digital Inputs/Channel 10
//     Task_P1 Inputs/IO.I107[11] <-> I107 (GSIO-A-16DIN)/Digital Inputs/Channel 11
//     Task_P1 Inputs/IO.I107[12] <-> I107 (GSIO-A-16DIN)/Digital Inputs/Channel 12
//     Task_P1 Inputs/IO.I107[13] <-> I107 (GSIO-A-16DIN)/Digital Inputs/Channel 13
//     Task_P1 Inputs/IO.I107[14] <-> I107 (GSIO-A-16DIN)/Digital Inputs/Channel 14
//     Task_P1 Inputs/IO.I107[15] <-> I107 (GSIO-A-16DIN)/Digital Inputs/Channel 15
//     Task_P1 Inputs/IO.I107[16] <-> I107 (GSIO-A-16DIN)/Digital Inputs/Channel 16
//     Task_P1 Inputs/IO.I107[1] <-> I107 (GSIO-A-16DIN)/Digital Inputs/Channel 1
//     Task_P1 Inputs/IO.I107[2] <-> I107 (GSIO-A-16DIN)/Digital Inputs/Channel 2
//     Task_P1 Inputs/IO.I107[3] <-> I107 (GSIO-A-16DIN)/Digital Inputs/Channel 3
//     Task_P1 Inputs/IO.I107[4] <-> I107 (GSIO-A-16DIN)/Digital Inputs/Channel 4
//     Task_P1 Inputs/IO.I107[5] <-> I107 (GSIO-A-16DIN)/Digital Inputs/Channel 5
//     Task_P1 Inputs/IO.I107[6] <-> I107 (GSIO-A-16DIN)/Digital Inputs/Channel 6
//     Task_P1 Inputs/IO.I107[7] <-> I107 (GSIO-A-16DIN)/Digital Inputs/Channel 7
//     Task_P1 Inputs/IO.I107[8] <-> I107 (GSIO-A-16DIN)/Digital Inputs/Channel 8
//     Task_P1 Inputs/IO.I107[9] <-> I107 (GSIO-A-16DIN)/Digital Inputs/Channel 9
//     Task_P1 Inputs/IO.I108[10] <-> I108 (GSIO-A-16DIN)/Digital Inputs/Channel 10
//     Task_P1 Inputs/IO.I108[11] <-> I108 (GSIO-A-16DIN)/Digital Inputs/Channel 11
//     Task_P1 Inputs/IO.I108[12] <-> I108 (GSIO-A-16DIN)/Digital Inputs/Channel 12
//     Task_P1 Inputs/IO.I108[13] <-> I108 (GSIO-A-16DIN)/Digital Inputs/Channel 13
//     Task_P1 Inputs/IO.I108[14] <-> I108 (GSIO-A-16DIN)/Digital Inputs/Channel 14
//     Task_P1 Inputs/IO.I108[15] <-> I108 (GSIO-A-16DIN)/Digital Inputs/Channel 15
//     Task_P1 Inputs/IO.I108[16] <-> I108 (GSIO-A-16DIN)/Digital Inputs/Channel 16
//     Task_P1 Inputs/IO.I108[1] <-> I108 (GSIO-A-16DIN)/Digital Inputs/Channel 1
//     Task_P1 Inputs/IO.I108[2] <-> I108 (GSIO-A-16DIN)/Digital Inputs/Channel 2
//     Task_P1 Inputs/IO.I108[3] <-> I108 (GSIO-A-16DIN)/Digital Inputs/Channel 3
//     Task_P1 Inputs/IO.I108[4] <-> I108 (GSIO-A-16DIN)/Digital Inputs/Channel 4
//     Task_P1 Inputs/IO.I108[5] <-> I108 (GSIO-A-16DIN)/Digital Inputs/Channel 5
//     Task_P1 Inputs/IO.I108[6] <-> I108 (GSIO-A-16DIN)/Digital Inputs/Channel 6
//     Task_P1 Inputs/IO.I108[7] <-> I108 (GSIO-A-16DIN)/Digital Inputs/Channel 7
//     Task_P1 Inputs/IO.I108[8] <-> I108 (GSIO-A-16DIN)/Digital Inputs/Channel 8
//     Task_P1 Inputs/IO.I108[9] <-> I108 (GSIO-A-16DIN)/Digital Inputs/Channel 9
//     Task_P1 Inputs/IO.I109[10] <-> I109 (GSIO-A-16DIN)/Digital Inputs/Channel 10
//     Task_P1 Inputs/IO.I109[11] <-> I109 (GSIO-A-16DIN)/Digital Inputs/Channel 11
//     Task_P1 Inputs/IO.I109[12] <-> I109 (GSIO-A-16DIN)/Digital Inputs/Channel 12
//     Task_P1 Inputs/IO.I109[13] <-> I109 (GSIO-A-16DIN)/Digital Inputs/Channel 13
//     Task_P1 Inputs/IO.I109[14] <-> I109 (GSIO-A-16DIN)/Digital Inputs/Channel 14
//     Task_P1 Inputs/IO.I109[15] <-> I109 (GSIO-A-16DIN)/Digital Inputs/Channel 15
//     Task_P1 Inputs/IO.I109[16] <-> I109 (GSIO-A-16DIN)/Digital Inputs/Channel 16
//     Task_P1 Inputs/IO.I109[1] <-> I109 (GSIO-A-16DIN)/Digital Inputs/Channel 1
//     Task_P1 Inputs/IO.I109[2] <-> I109 (GSIO-A-16DIN)/Digital Inputs/Channel 2
//     Task_P1 Inputs/IO.I109[3] <-> I109 (GSIO-A-16DIN)/Digital Inputs/Channel 3
//     Task_P1 Inputs/IO.I109[4] <-> I109 (GSIO-A-16DIN)/Digital Inputs/Channel 4
//     Task_P1 Inputs/IO.I109[5] <-> I109 (GSIO-A-16DIN)/Digital Inputs/Channel 5
//     Task_P1 Inputs/IO.I109[6] <-> I109 (GSIO-A-16DIN)/Digital Inputs/Channel 6
//     Task_P1 Inputs/IO.I109[7] <-> I109 (GSIO-A-16DIN)/Digital Inputs/Channel 7
//     Task_P1 Inputs/IO.I109[8] <-> I109 (GSIO-A-16DIN)/Digital Inputs/Channel 8
//     Task_P1 Inputs/IO.I109[9] <-> I109 (GSIO-A-16DIN)/Digital Inputs/Channel 9
//     Task_P1 Outputs/IO.AO101[{0..3}] <-> AO101 (GSIO-A-4AOV)/Analog Outputs/Channel {1..4}  (4 links)
//     Task_P1 Outputs/IO.Q101[10] <-> Q101 (GSIO-A-16DON)/Digital Outputs/Channel 10
//     Task_P1 Outputs/IO.Q101[11] <-> Q101 (GSIO-A-16DON)/Digital Outputs/Channel 11
//     Task_P1 Outputs/IO.Q101[12] <-> Q101 (GSIO-A-16DON)/Digital Outputs/Channel 12
//     Task_P1 Outputs/IO.Q101[13] <-> Q101 (GSIO-A-16DON)/Digital Outputs/Channel 13
//     Task_P1 Outputs/IO.Q101[14] <-> Q101 (GSIO-A-16DON)/Digital Outputs/Channel 14
//     Task_P1 Outputs/IO.Q101[15] <-> Q101 (GSIO-A-16DON)/Digital Outputs/Channel 15
//     Task_P1 Outputs/IO.Q101[16] <-> Q101 (GSIO-A-16DON)/Digital Outputs/Channel 16
//     Task_P1 Outputs/IO.Q101[1] <-> Q101 (GSIO-A-16DON)/Digital Outputs/Channel 1
//     Task_P1 Outputs/IO.Q101[2] <-> Q101 (GSIO-A-16DON)/Digital Outputs/Channel 2
//     Task_P1 Outputs/IO.Q101[3] <-> Q101 (GSIO-A-16DON)/Digital Outputs/Channel 3
//     Task_P1 Outputs/IO.Q101[4] <-> Q101 (GSIO-A-16DON)/Digital Outputs/Channel 4
//     Task_P1 Outputs/IO.Q101[5] <-> Q101 (GSIO-A-16DON)/Digital Outputs/Channel 5
//     Task_P1 Outputs/IO.Q101[6] <-> Q101 (GSIO-A-16DON)/Digital Outputs/Channel 6
//     Task_P1 Outputs/IO.Q101[7] <-> Q101 (GSIO-A-16DON)/Digital Outputs/Channel 7
//     Task_P1 Outputs/IO.Q101[8] <-> Q101 (GSIO-A-16DON)/Digital Outputs/Channel 8
//     Task_P1 Outputs/IO.Q101[9] <-> Q101 (GSIO-A-16DON)/Digital Outputs/Channel 9
//     Task_P1 Outputs/IO.Q102[10] <-> Q102 (GSIO-A-16DON)/Digital Outputs/Channel 10
//     Task_P1 Outputs/IO.Q102[11] <-> Q102 (GSIO-A-16DON)/Digital Outputs/Channel 11
//     Task_P1 Outputs/IO.Q102[12] <-> Q102 (GSIO-A-16DON)/Digital Outputs/Channel 12
//     Task_P1 Outputs/IO.Q102[13] <-> Q102 (GSIO-A-16DON)/Digital Outputs/Channel 13
//     Task_P1 Outputs/IO.Q102[14] <-> Q102 (GSIO-A-16DON)/Digital Outputs/Channel 14
//     Task_P1 Outputs/IO.Q102[15] <-> Q102 (GSIO-A-16DON)/Digital Outputs/Channel 15
//     Task_P1 Outputs/IO.Q102[16] <-> Q102 (GSIO-A-16DON)/Digital Outputs/Channel 16
//     Task_P1 Outputs/IO.Q102[1] <-> Q102 (GSIO-A-16DON)/Digital Outputs/Channel 1
//     Task_P1 Outputs/IO.Q102[2] <-> Q102 (GSIO-A-16DON)/Digital Outputs/Channel 2
//     Task_P1 Outputs/IO.Q102[3] <-> Q102 (GSIO-A-16DON)/Digital Outputs/Channel 3
//     Task_P1 Outputs/IO.Q102[4] <-> Q102 (GSIO-A-16DON)/Digital Outputs/Channel 4
//     Task_P1 Outputs/IO.Q102[5] <-> Q102 (GSIO-A-16DON)/Digital Outputs/Channel 5
//     Task_P1 Outputs/IO.Q102[6] <-> Q102 (GSIO-A-16DON)/Digital Outputs/Channel 6
//     Task_P1 Outputs/IO.Q102[7] <-> Q102 (GSIO-A-16DON)/Digital Outputs/Channel 7
//     Task_P1 Outputs/IO.Q102[8] <-> Q102 (GSIO-A-16DON)/Digital Outputs/Channel 8
//     Task_P1 Outputs/IO.Q102[9] <-> Q102 (GSIO-A-16DON)/Digital Outputs/Channel 9
//     Task_P1 Outputs/IO.Q103[10] <-> Q103 (GSIO-A-16DON)/Digital Outputs/Channel 10
//     Task_P1 Outputs/IO.Q103[11] <-> Q103 (GSIO-A-16DON)/Digital Outputs/Channel 11
//     Task_P1 Outputs/IO.Q103[12] <-> Q103 (GSIO-A-16DON)/Digital Outputs/Channel 12
//     Task_P1 Outputs/IO.Q103[13] <-> Q103 (GSIO-A-16DON)/Digital Outputs/Channel 13
//     Task_P1 Outputs/IO.Q103[14] <-> Q103 (GSIO-A-16DON)/Digital Outputs/Channel 14
//     Task_P1 Outputs/IO.Q103[15] <-> Q103 (GSIO-A-16DON)/Digital Outputs/Channel 15
//     Task_P1 Outputs/IO.Q103[16] <-> Q103 (GSIO-A-16DON)/Digital Outputs/Channel 16
//     Task_P1 Outputs/IO.Q103[1] <-> Q103 (GSIO-A-16DON)/Digital Outputs/Channel 1
//     Task_P1 Outputs/IO.Q103[2] <-> Q103 (GSIO-A-16DON)/Digital Outputs/Channel 2
//     Task_P1 Outputs/IO.Q103[3] <-> Q103 (GSIO-A-16DON)/Digital Outputs/Channel 3
//     Task_P1 Outputs/IO.Q103[4] <-> Q103 (GSIO-A-16DON)/Digital Outputs/Channel 4
//     Task_P1 Outputs/IO.Q103[5] <-> Q103 (GSIO-A-16DON)/Digital Outputs/Channel 5
//     Task_P1 Outputs/IO.Q103[6] <-> Q103 (GSIO-A-16DON)/Digital Outputs/Channel 6
//     Task_P1 Outputs/IO.Q103[7] <-> Q103 (GSIO-A-16DON)/Digital Outputs/Channel 7
//     Task_P1 Outputs/IO.Q103[8] <-> Q103 (GSIO-A-16DON)/Digital Outputs/Channel 8
//     Task_P1 Outputs/IO.Q103[9] <-> Q103 (GSIO-A-16DON)/Digital Outputs/Channel 9
//     Task_P1 Outputs/IO.Q104[10] <-> Q104 (GSIO-A-16DON)/Digital Outputs/Channel 10
//     Task_P1 Outputs/IO.Q104[11] <-> Q104 (GSIO-A-16DON)/Digital Outputs/Channel 11
//     Task_P1 Outputs/IO.Q104[12] <-> Q104 (GSIO-A-16DON)/Digital Outputs/Channel 12
//     Task_P1 Outputs/IO.Q104[13] <-> Q104 (GSIO-A-16DON)/Digital Outputs/Channel 13
//     Task_P1 Outputs/IO.Q104[14] <-> Q104 (GSIO-A-16DON)/Digital Outputs/Channel 14
//     Task_P1 Outputs/IO.Q104[15] <-> Q104 (GSIO-A-16DON)/Digital Outputs/Channel 15
//     Task_P1 Outputs/IO.Q104[16] <-> Q104 (GSIO-A-16DON)/Digital Outputs/Channel 16
//     Task_P1 Outputs/IO.Q104[1] <-> Q104 (GSIO-A-16DON)/Digital Outputs/Channel 1
//     Task_P1 Outputs/IO.Q104[2] <-> Q104 (GSIO-A-16DON)/Digital Outputs/Channel 2
//     Task_P1 Outputs/IO.Q104[3] <-> Q104 (GSIO-A-16DON)/Digital Outputs/Channel 3
//     Task_P1 Outputs/IO.Q104[4] <-> Q104 (GSIO-A-16DON)/Digital Outputs/Channel 4
//     Task_P1 Outputs/IO.Q104[5] <-> Q104 (GSIO-A-16DON)/Digital Outputs/Channel 5
//     Task_P1 Outputs/IO.Q104[6] <-> Q104 (GSIO-A-16DON)/Digital Outputs/Channel 6
//     Task_P1 Outputs/IO.Q104[7] <-> Q104 (GSIO-A-16DON)/Digital Outputs/Channel 7
//     Task_P1 Outputs/IO.Q104[8] <-> Q104 (GSIO-A-16DON)/Digital Outputs/Channel 8
//     Task_P1 Outputs/IO.Q104[9] <-> Q104 (GSIO-A-16DON)/Digital Outputs/Channel 9
//     Task_P1 Outputs/IO.Q105[10] <-> Q105 (GSIO-A-16DON)/Digital Outputs/Channel 10
//     Task_P1 Outputs/IO.Q105[11] <-> Q105 (GSIO-A-16DON)/Digital Outputs/Channel 11
//     Task_P1 Outputs/IO.Q105[12] <-> Q105 (GSIO-A-16DON)/Digital Outputs/Channel 12
//     Task_P1 Outputs/IO.Q105[13] <-> Q105 (GSIO-A-16DON)/Digital Outputs/Channel 13
//     Task_P1 Outputs/IO.Q105[14] <-> Q105 (GSIO-A-16DON)/Digital Outputs/Channel 14
//     Task_P1 Outputs/IO.Q105[15] <-> Q105 (GSIO-A-16DON)/Digital Outputs/Channel 15
//     Task_P1 Outputs/IO.Q105[16] <-> Q105 (GSIO-A-16DON)/Digital Outputs/Channel 16
//     Task_P1 Outputs/IO.Q105[1] <-> Q105 (GSIO-A-16DON)/Digital Outputs/Channel 1
//     Task_P1 Outputs/IO.Q105[2] <-> Q105 (GSIO-A-16DON)/Digital Outputs/Channel 2
//     Task_P1 Outputs/IO.Q105[3] <-> Q105 (GSIO-A-16DON)/Digital Outputs/Channel 3
//     Task_P1 Outputs/IO.Q105[4] <-> Q105 (GSIO-A-16DON)/Digital Outputs/Channel 4
//     Task_P1 Outputs/IO.Q105[5] <-> Q105 (GSIO-A-16DON)/Digital Outputs/Channel 5
//     Task_P1 Outputs/IO.Q105[6] <-> Q105 (GSIO-A-16DON)/Digital Outputs/Channel 6
//     Task_P1 Outputs/IO.Q105[7] <-> Q105 (GSIO-A-16DON)/Digital Outputs/Channel 7
//     Task_P1 Outputs/IO.Q105[8] <-> Q105 (GSIO-A-16DON)/Digital Outputs/Channel 8
//     Task_P1 Outputs/IO.Q105[9] <-> Q105 (GSIO-A-16DON)/Digital Outputs/Channel 9
//     Task_P1 Outputs/IO.Q106[10] <-> Q106 (GSIO-A-16DON)/Digital Outputs/Channel 10
//     Task_P1 Outputs/IO.Q106[11] <-> Q106 (GSIO-A-16DON)/Digital Outputs/Channel 11
//     Task_P1 Outputs/IO.Q106[12] <-> Q106 (GSIO-A-16DON)/Digital Outputs/Channel 12
//     Task_P1 Outputs/IO.Q106[13] <-> Q106 (GSIO-A-16DON)/Digital Outputs/Channel 13
//     Task_P1 Outputs/IO.Q106[14] <-> Q106 (GSIO-A-16DON)/Digital Outputs/Channel 14
//     Task_P1 Outputs/IO.Q106[15] <-> Q106 (GSIO-A-16DON)/Digital Outputs/Channel 15
//     Task_P1 Outputs/IO.Q106[16] <-> Q106 (GSIO-A-16DON)/Digital Outputs/Channel 16
//     Task_P1 Outputs/IO.Q106[1] <-> Q106 (GSIO-A-16DON)/Digital Outputs/Channel 1
//     Task_P1 Outputs/IO.Q106[2] <-> Q106 (GSIO-A-16DON)/Digital Outputs/Channel 2
//     Task_P1 Outputs/IO.Q106[3] <-> Q106 (GSIO-A-16DON)/Digital Outputs/Channel 3
//     Task_P1 Outputs/IO.Q106[4] <-> Q106 (GSIO-A-16DON)/Digital Outputs/Channel 4
//     Task_P1 Outputs/IO.Q106[5] <-> Q106 (GSIO-A-16DON)/Digital Outputs/Channel 5
//     Task_P1 Outputs/IO.Q106[6] <-> Q106 (GSIO-A-16DON)/Digital Outputs/Channel 6
//     Task_P1 Outputs/IO.Q106[7] <-> Q106 (GSIO-A-16DON)/Digital Outputs/Channel 7
//     Task_P1 Outputs/IO.Q106[8] <-> Q106 (GSIO-A-16DON)/Digital Outputs/Channel 8
//     Task_P1 Outputs/IO.Q106[9] <-> Q106 (GSIO-A-16DON)/Digital Outputs/Channel 9
//     Task_P1 Outputs/IO.Q107[10] <-> Q107 (GSIO-A-16DON)/Digital Outputs/Channel 10
//     Task_P1 Outputs/IO.Q107[11] <-> Q107 (GSIO-A-16DON)/Digital Outputs/Channel 11
//     Task_P1 Outputs/IO.Q107[12] <-> Q107 (GSIO-A-16DON)/Digital Outputs/Channel 12
//     Task_P1 Outputs/IO.Q107[13] <-> Q107 (GSIO-A-16DON)/Digital Outputs/Channel 13
//     Task_P1 Outputs/IO.Q107[14] <-> Q107 (GSIO-A-16DON)/Digital Outputs/Channel 14
//     Task_P1 Outputs/IO.Q107[15] <-> Q107 (GSIO-A-16DON)/Digital Outputs/Channel 15
//     Task_P1 Outputs/IO.Q107[16] <-> Q107 (GSIO-A-16DON)/Digital Outputs/Channel 16
//     Task_P1 Outputs/IO.Q107[1] <-> Q107 (GSIO-A-16DON)/Digital Outputs/Channel 1
//     Task_P1 Outputs/IO.Q107[2] <-> Q107 (GSIO-A-16DON)/Digital Outputs/Channel 2
//     Task_P1 Outputs/IO.Q107[3] <-> Q107 (GSIO-A-16DON)/Digital Outputs/Channel 3
//     Task_P1 Outputs/IO.Q107[4] <-> Q107 (GSIO-A-16DON)/Digital Outputs/Channel 4
//     Task_P1 Outputs/IO.Q107[5] <-> Q107 (GSIO-A-16DON)/Digital Outputs/Channel 5
//     Task_P1 Outputs/IO.Q107[6] <-> Q107 (GSIO-A-16DON)/Digital Outputs/Channel 6
//     Task_P1 Outputs/IO.Q107[7] <-> Q107 (GSIO-A-16DON)/Digital Outputs/Channel 7
//     Task_P1 Outputs/IO.Q107[8] <-> Q107 (GSIO-A-16DON)/Digital Outputs/Channel 8
//     Task_P1 Outputs/IO.Q107[9] <-> Q107 (GSIO-A-16DON)/Digital Outputs/Channel 9
//     Task_P1 Outputs/IO.Q108[10] <-> Q108 (GSIO-A-16DON)/Digital Outputs/Channel 10
//     Task_P1 Outputs/IO.Q108[11] <-> Q108 (GSIO-A-16DON)/Digital Outputs/Channel 11
//     Task_P1 Outputs/IO.Q108[12] <-> Q108 (GSIO-A-16DON)/Digital Outputs/Channel 12
//     Task_P1 Outputs/IO.Q108[13] <-> Q108 (GSIO-A-16DON)/Digital Outputs/Channel 13
//     Task_P1 Outputs/IO.Q108[14] <-> Q108 (GSIO-A-16DON)/Digital Outputs/Channel 14
//     Task_P1 Outputs/IO.Q108[15] <-> Q108 (GSIO-A-16DON)/Digital Outputs/Channel 15
//     Task_P1 Outputs/IO.Q108[16] <-> Q108 (GSIO-A-16DON)/Digital Outputs/Channel 16
//     Task_P1 Outputs/IO.Q108[1] <-> Q108 (GSIO-A-16DON)/Digital Outputs/Channel 1
//     Task_P1 Outputs/IO.Q108[2] <-> Q108 (GSIO-A-16DON)/Digital Outputs/Channel 2
//     Task_P1 Outputs/IO.Q108[3] <-> Q108 (GSIO-A-16DON)/Digital Outputs/Channel 3
//     Task_P1 Outputs/IO.Q108[4] <-> Q108 (GSIO-A-16DON)/Digital Outputs/Channel 4
//     Task_P1 Outputs/IO.Q108[5] <-> Q108 (GSIO-A-16DON)/Digital Outputs/Channel 5
//     Task_P1 Outputs/IO.Q108[6] <-> Q108 (GSIO-A-16DON)/Digital Outputs/Channel 6
//     Task_P1 Outputs/IO.Q108[7] <-> Q108 (GSIO-A-16DON)/Digital Outputs/Channel 7
//     Task_P1 Outputs/IO.Q108[8] <-> Q108 (GSIO-A-16DON)/Digital Outputs/Channel 8
//     Task_P1 Outputs/IO.Q108[9] <-> Q108 (GSIO-A-16DON)/Digital Outputs/Channel 9
//     Task_P1 Outputs/IO.Q109[10] <-> Q109 (GSIO-A-16DON)/Digital Outputs/Channel 10
//     Task_P1 Outputs/IO.Q109[11] <-> Q109 (GSIO-A-16DON)/Digital Outputs/Channel 11
//     Task_P1 Outputs/IO.Q109[12] <-> Q109 (GSIO-A-16DON)/Digital Outputs/Channel 12
//     Task_P1 Outputs/IO.Q109[13] <-> Q109 (GSIO-A-16DON)/Digital Outputs/Channel 13
//     Task_P1 Outputs/IO.Q109[14] <-> Q109 (GSIO-A-16DON)/Digital Outputs/Channel 14
//     Task_P1 Outputs/IO.Q109[15] <-> Q109 (GSIO-A-16DON)/Digital Outputs/Channel 15
//     Task_P1 Outputs/IO.Q109[16] <-> Q109 (GSIO-A-16DON)/Digital Outputs/Channel 16
//     Task_P1 Outputs/IO.Q109[1] <-> Q109 (GSIO-A-16DON)/Digital Outputs/Channel 1
//     Task_P1 Outputs/IO.Q109[2] <-> Q109 (GSIO-A-16DON)/Digital Outputs/Channel 2
//     Task_P1 Outputs/IO.Q109[3] <-> Q109 (GSIO-A-16DON)/Digital Outputs/Channel 3
//     Task_P1 Outputs/IO.Q109[4] <-> Q109 (GSIO-A-16DON)/Digital Outputs/Channel 4
//     Task_P1 Outputs/IO.Q109[5] <-> Q109 (GSIO-A-16DON)/Digital Outputs/Channel 5
//     Task_P1 Outputs/IO.Q109[6] <-> Q109 (GSIO-A-16DON)/Digital Outputs/Channel 6
//     Task_P1 Outputs/IO.Q109[7] <-> Q109 (GSIO-A-16DON)/Digital Outputs/Channel 7
//     Task_P1 Outputs/IO.Q109[8] <-> Q109 (GSIO-A-16DON)/Digital Outputs/Channel 8
//     Task_P1 Outputs/IO.Q109[9] <-> Q109 (GSIO-A-16DON)/Digital Outputs/Channel 9
//   MQPLC/MQPLC Instance <-> Device 3 (EtherCAT)/Box 2 (CU1128)/正极上表面除尘皮带(InoSV660N)
//     Task_P1 Inputs/GMotion.DrivesOP[18] <-> InfoData/State
//     Task_P1 Inputs/GMotion.arrAxisCtrl[18].Io.DigitalInputs <-> Inputs/Digital inputs
//     Task_P1 Inputs/GMotion.arrAxisCtrl[18].Io.ErrorCode <-> Inputs/Error code
//     Task_P1 Inputs/GMotion.iActTorque_M[18] <-> Inputs/Torque actual value
//   MQPLC/MQPLC Instance <-> Device 3 (EtherCAT)/Box 2 (CU1128)/正极下表面除尘倒装皮带(InoSV660N)
//     Task_P1 Inputs/GMotion.DrivesOP[19] <-> InfoData/State
//     Task_P1 Inputs/GMotion.arrAxisCtrl[19].Io.DigitalInputs <-> Inputs/Digital inputs
//     Task_P1 Inputs/GMotion.arrAxisCtrl[19].Io.ErrorCode <-> Inputs/Error code
//     Task_P1 Inputs/GMotion.iActTorque_M[19] <-> Inputs/Torque actual value
//   MQPLC/MQPLC Instance <-> Device 3 (EtherCAT)/Box 2 (CU1128)/正极倒角模具(InoSV660N)
//     Task_P1 Inputs/GMotion.DrivesOP[6] <-> InfoData/State
//     Task_P1 Inputs/GMotion.arrAxisCtrl[6].Io.DigitalInputs <-> Inputs/Digital inputs
//     Task_P1 Inputs/GMotion.arrAxisCtrl[6].Io.ErrorCode <-> Inputs/Error code
//     Task_P1 Inputs/GMotion.iActTorque_M[6] <-> Inputs/Torque actual value
//   MQPLC/MQPLC Instance <-> Device 3 (EtherCAT)/Box 2 (CU1128)/正极右放卷电机(InoSV660N)
//     Task_P1 Inputs/GMotion.DrivesOP[2] <-> InfoData/State
//     Task_P1 Inputs/GMotion.arrAxisCtrl[2].Io.DigitalInputs <-> Inputs/Digital inputs
//     Task_P1 Inputs/GMotion.arrAxisCtrl[2].Io.ErrorCode <-> Inputs/Error code
//     Task_P1 Inputs/GMotion.iActTorque_M[2] <-> Inputs/Torque actual value
//   MQPLC/MQPLC Instance <-> Device 3 (EtherCAT)/Box 2 (CU1128)/正极尺寸CCD压片升降(InoSV660N)
//     Task_P1 Inputs/GMotion.DrivesOP[14] <-> InfoData/State
//     Task_P1 Inputs/GMotion.arrAxisCtrl[14].Io.DigitalInputs <-> Inputs/Digital inputs
//     Task_P1 Inputs/GMotion.arrAxisCtrl[14].Io.ErrorCode <-> Inputs/Error code
//     Task_P1 Inputs/GMotion.iActTorque_M[14] <-> Inputs/Torque actual value
//   MQPLC/MQPLC Instance <-> Device 3 (EtherCAT)/Box 2 (CU1128)/正极左放卷电机(InoSV660N)
//     Task_P1 Inputs/GMotion.DrivesOP[1] <-> InfoData/State
//     Task_P1 Inputs/GMotion.arrAxisCtrl[1].Io.DigitalInputs <-> Inputs/Digital inputs
//     Task_P1 Inputs/GMotion.arrAxisCtrl[1].Io.ErrorCode <-> Inputs/Error code
//     Task_P1 Inputs/GMotion.iActTorque_M[1] <-> Inputs/Torque actual value
//   MQPLC/MQPLC Instance <-> Device 3 (EtherCAT)/Box 2 (CU1128)/正极模具纠偏X轴(肩宽)(InoSV660N)
//     Task_P1 Inputs/GMotion.DrivesOP[7] <-> InfoData/State
//     Task_P1 Inputs/GMotion.arrAxisCtrl[7].Io.DigitalInputs <-> Inputs/Digital inputs
//     Task_P1 Inputs/GMotion.arrAxisCtrl[7].Io.ErrorCode <-> Inputs/Error code
//     Task_P1 Inputs/GMotion.iActTorque_M[7] <-> Inputs/Torque actual value
//   MQPLC/MQPLC Instance <-> Device 3 (EtherCAT)/Box 2 (CU1128)/正极模具纠偏Y轴(InoSV660N)
//     Task_P1 Inputs/GMotion.DrivesOP[8] <-> InfoData/State
//     Task_P1 Inputs/GMotion.arrAxisCtrl[8].Io.DigitalInputs <-> Inputs/Digital inputs
//     Task_P1 Inputs/GMotion.arrAxisCtrl[8].Io.ErrorCode <-> Inputs/Error code
//     Task_P1 Inputs/GMotion.iActTorque_M[8] <-> Inputs/Torque actual value
//   MQPLC/MQPLC Instance <-> Device 3 (EtherCAT)/Box 2 (CU1128)/正极模切主驱动(CDHD)
//     Task_P1 Inputs/GMotion.DrivesOP[9] <-> InfoData/State
//     Task_P1 Inputs/GMotion.arrAxisCtrl[9].Io.DigitalInputs <-> TxPDO 4/Digital inputs
//     Task_P1 Inputs/GMotion.iActTorque_M[9] <-> TxPDO 1/Torque Actual Value
//   MQPLC/MQPLC Instance <-> Device 3 (EtherCAT)/Box 2 (CU1128)/正极模切前摆杆张力(InoSV660N)
//     Task_P1 Inputs/GMotion.DrivesOP[3] <-> InfoData/State
//     Task_P1 Inputs/GMotion.arrAxisCtrl[3].Io.DigitalInputs <-> Inputs/Digital inputs
//     Task_P1 Inputs/GMotion.arrAxisCtrl[3].Io.ErrorCode <-> Inputs/Error code
//     Task_P1 Inputs/GMotion.iActDriveTorque[1] <-> Inputs/Torque actual value
//     Task_P1 Outputs/GMotion.iMaxProfileVelo[1] <-> Outputs/Max profile velocity
//     Task_P1 Outputs/GMotion.iNegtiveTorqueLimits[1] <-> Outputs/Negative torque limit value
//     Task_P1 Outputs/GMotion.iPostiveTorqueLimits[1] <-> Outputs/Positive torque limit value
//     Task_P1 Outputs/GMotion.iSetDriveMode[1] <-> Outputs/Modes of operation
//     Task_P1 Outputs/GMotion.iTargetTorque[1] <-> Outputs/Target torque
//   MQPLC/MQPLC Instance <-> Device 3 (EtherCAT)/Box 2 (CU1128)/正极模切极片缓存(CDHD)
//     Task_P1 Inputs/GMotion.DrivesOP[5] <-> InfoData/State
//     Task_P1 Inputs/GMotion.arrAxisCtrl[5].Io.DigitalInputs <-> TxPDO 4/Digital inputs
//     Task_P1 Inputs/GMotion.iActTorque_M[5] <-> TxPDO 1/Torque Actual Value
//   MQPLC/MQPLC Instance <-> Device 3 (EtherCAT)/Box 2 (CU1128)/正极模切辅助驱动(InoSV660N)
//     Task_P1 Inputs/GMotion.DrivesOP[4] <-> InfoData/State
//     Task_P1 Inputs/GMotion.arrAxisCtrl[4].Io.DigitalInputs <-> Inputs/Digital inputs
//     Task_P1 Inputs/GMotion.arrAxisCtrl[4].Io.ErrorCode <-> Inputs/Error code
//     Task_P1 Inputs/GMotion.iActTorque_M[4] <-> Inputs/Torque actual value
//   MQPLC/MQPLC Instance <-> Device 3 (EtherCAT)/Box 2 (CU1128)/正极裁切切刀(InoSV660N)
//     Task_P1 Inputs/GMotion.DrivesOP[10] <-> InfoData/State
//     Task_P1 Inputs/GMotion.arrAxisCtrl[10].Io.DigitalInputs <-> Inputs/Digital inputs
//     Task_P1 Inputs/GMotion.arrAxisCtrl[10].Io.ErrorCode <-> Inputs/Error code
//     Task_P1 Inputs/GMotion.iActTorque_M[10] <-> Inputs/Torque actual value
//   MQPLC/MQPLC Instance <-> Device 3 (EtherCAT)/Box 2 (CU1128)/正极裁切角度纠偏(InoSV660N)
//     Task_P1 Inputs/GMotion.DrivesOP[11] <-> InfoData/State
//     Task_P1 Inputs/GMotion.arrAxisCtrl[11].Io.DigitalInputs <-> Inputs/Digital inputs
//     Task_P1 Inputs/GMotion.arrAxisCtrl[11].Io.ErrorCode <-> Inputs/Error code
//     Task_P1 Inputs/GMotion.iActTorque_M[11] <-> Inputs/Torque actual value
//   MQPLC/MQPLC Instance <-> Device 3 (EtherCAT)/Box 2 (CU1128)/正极裁切输送带换型(InoSV660N)
//     Task_P1 Inputs/GMotion.DrivesOP[13] <-> InfoData/State
//     Task_P1 Inputs/GMotion.arrAxisCtrl[13].Io.DigitalInputs <-> Inputs/Digital inputs
//     Task_P1 Inputs/GMotion.arrAxisCtrl[13].Io.ErrorCode <-> Inputs/Error code
//     Task_P1 Inputs/GMotion.iActTorque_M[13] <-> Inputs/Torque actual value
//   MQPLC/MQPLC Instance <-> Device 3 (EtherCAT)/Box 2 (CU1128)/正极裁切输送皮带(InoSV660N)
//     Task_P1 Inputs/GMotion.DrivesOP[12] <-> InfoData/State
//     Task_P1 Inputs/GMotion.arrAxisCtrl[12].Io.DigitalInputs <-> Inputs/Digital inputs
//     Task_P1 Inputs/GMotion.arrAxisCtrl[12].Io.ErrorCode <-> Inputs/Error code
//     Task_P1 Inputs/GMotion.iActTorque_M[12] <-> Inputs/Torque actual value
//   MQPLC/MQPLC Instance <-> Device 3 (EtherCAT)/Box 2 (CU1128)/正极踢单张废料(InoSV660N)
//     Task_P1 Inputs/GMotion.DrivesOP[17] <-> InfoData/State
//     Task_P1 Inputs/GMotion.arrAxisCtrl[17].Io.DigitalInputs <-> Inputs/Digital inputs
//     Task_P1 Inputs/GMotion.arrAxisCtrl[17].Io.ErrorCode <-> Inputs/Error code
//     Task_P1 Inputs/GMotion.iActTorque_M[17] <-> Inputs/Torque actual value
//   MQPLC/MQPLC Instance <-> Device 3 (EtherCAT)/Box 2 (CU1128)/正极踢废倒装皮带(InoSV660N)
//     Task_P1 Inputs/GMotion.DrivesOP[15] <-> InfoData/State
//     Task_P1 Inputs/GMotion.arrAxisCtrl[15].Io.DigitalInputs <-> Inputs/Digital inputs
//     Task_P1 Inputs/GMotion.arrAxisCtrl[15].Io.ErrorCode <-> Inputs/Error code
//     Task_P1 Inputs/GMotion.iActTorque_M[15] <-> Inputs/Torque actual value
//   MQPLC/MQPLC Instance <-> Device 3 (EtherCAT)/Box 2 (CU1128)/正极踢连续废料(InoSV660N)
//     Task_P1 Inputs/GMotion.DrivesOP[16] <-> InfoData/State
//     Task_P1 Inputs/GMotion.arrAxisCtrl[16].Io.DigitalInputs <-> Inputs/Digital inputs
//     Task_P1 Inputs/GMotion.arrAxisCtrl[16].Io.ErrorCode <-> Inputs/Error code
//     Task_P1 Inputs/GMotion.iActTorque_M[16] <-> Inputs/Torque actual value
//   MQPLC/MQPLC Instance <-> Device 3 (EtherCAT)/Box 2 (CU1128)/负极IO耦合器(GSIO-A-ECC)
//     Task_P1 Inputs/IO.AI201[0] <-> AI201 (GSIO-A-4AIHV)/Analog Inputs/Channel 1
//     Task_P1 Inputs/IO.AI201[1] <-> AI201 (GSIO-A-4AIHV)/Analog Inputs/Channel 2
//     Task_P1 Inputs/IO.AI201[2] <-> AI201 (GSIO-A-4AIHV)/Analog Inputs/Channel 3
//     Task_P1 Inputs/IO.AI201[3] <-> AI201 (GSIO-A-4AIHV)/Analog Inputs/Channel 4
//     Task_P1 Inputs/IO.AI202[0] <-> AI202 (GSIO-A-4AIHV)/Analog Inputs/Channel 1
//     Task_P1 Inputs/IO.AI202[1] <-> AI202 (GSIO-A-4AIHV)/Analog Inputs/Channel 2
//     Task_P1 Inputs/IO.AI202[2] <-> AI202 (GSIO-A-4AIHV)/Analog Inputs/Channel 3
//     Task_P1 Inputs/IO.AI202[3] <-> AI202 (GSIO-A-4AIHV)/Analog Inputs/Channel 4
//     Task_P1 Inputs/IO.I201[10] <-> I201 (GSIO-A-16DIN)/Digital Inputs/Channel 10
//     Task_P1 Inputs/IO.I201[11] <-> I201 (GSIO-A-16DIN)/Digital Inputs/Channel 11
//     Task_P1 Inputs/IO.I201[12] <-> I201 (GSIO-A-16DIN)/Digital Inputs/Channel 12
//     Task_P1 Inputs/IO.I201[13] <-> I201 (GSIO-A-16DIN)/Digital Inputs/Channel 13
//     Task_P1 Inputs/IO.I201[14] <-> I201 (GSIO-A-16DIN)/Digital Inputs/Channel 14
//     Task_P1 Inputs/IO.I201[15] <-> I201 (GSIO-A-16DIN)/Digital Inputs/Channel 15
//     Task_P1 Inputs/IO.I201[16] <-> I201 (GSIO-A-16DIN)/Digital Inputs/Channel 16
//     Task_P1 Inputs/IO.I201[1] <-> I201 (GSIO-A-16DIN)/Digital Inputs/Channel 1
//     Task_P1 Inputs/IO.I201[2] <-> I201 (GSIO-A-16DIN)/Digital Inputs/Channel 2
//     Task_P1 Inputs/IO.I201[3] <-> I201 (GSIO-A-16DIN)/Digital Inputs/Channel 3
//     Task_P1 Inputs/IO.I201[4] <-> I201 (GSIO-A-16DIN)/Digital Inputs/Channel 4
//     Task_P1 Inputs/IO.I201[5] <-> I201 (GSIO-A-16DIN)/Digital Inputs/Channel 5
//     Task_P1 Inputs/IO.I201[6] <-> I201 (GSIO-A-16DIN)/Digital Inputs/Channel 6
//     Task_P1 Inputs/IO.I201[7] <-> I201 (GSIO-A-16DIN)/Digital Inputs/Channel 7
//     Task_P1 Inputs/IO.I201[8] <-> I201 (GSIO-A-16DIN)/Digital Inputs/Channel 8
//     Task_P1 Inputs/IO.I201[9] <-> I201 (GSIO-A-16DIN)/Digital Inputs/Channel 9
//     Task_P1 Inputs/IO.I202[10] <-> I202 (GSIO-A-16DIN)/Digital Inputs/Channel 10
//     Task_P1 Inputs/IO.I202[11] <-> I202 (GSIO-A-16DIN)/Digital Inputs/Channel 11
//     Task_P1 Inputs/IO.I202[12] <-> I202 (GSIO-A-16DIN)/Digital Inputs/Channel 12
//     Task_P1 Inputs/IO.I202[13] <-> I202 (GSIO-A-16DIN)/Digital Inputs/Channel 13
//     Task_P1 Inputs/IO.I202[14] <-> I202 (GSIO-A-16DIN)/Digital Inputs/Channel 14
//     Task_P1 Inputs/IO.I202[15] <-> I202 (GSIO-A-16DIN)/Digital Inputs/Channel 15
//     Task_P1 Inputs/IO.I202[16] <-> I202 (GSIO-A-16DIN)/Digital Inputs/Channel 16
//     Task_P1 Inputs/IO.I202[1] <-> I202 (GSIO-A-16DIN)/Digital Inputs/Channel 1
//     Task_P1 Inputs/IO.I202[2] <-> I202 (GSIO-A-16DIN)/Digital Inputs/Channel 2
//     Task_P1 Inputs/IO.I202[3] <-> I202 (GSIO-A-16DIN)/Digital Inputs/Channel 3
//     Task_P1 Inputs/IO.I202[4] <-> I202 (GSIO-A-16DIN)/Digital Inputs/Channel 4
//     Task_P1 Inputs/IO.I202[5] <-> I202 (GSIO-A-16DIN)/Digital Inputs/Channel 5
//     Task_P1 Inputs/IO.I202[6] <-> I202 (GSIO-A-16DIN)/Digital Inputs/Channel 6
//     Task_P1 Inputs/IO.I202[7] <-> I202 (GSIO-A-16DIN)/Digital Inputs/Channel 7
//     Task_P1 Inputs/IO.I202[8] <-> I202 (GSIO-A-16DIN)/Digital Inputs/Channel 8
//     Task_P1 Inputs/IO.I202[9] <-> I202 (GSIO-A-16DIN)/Digital Inputs/Channel 9
//     Task_P1 Inputs/IO.I203[10] <-> I203 (GSIO-A-16DIN)/Digital Inputs/Channel 10
//     Task_P1 Inputs/IO.I203[11] <-> I203 (GSIO-A-16DIN)/Digital Inputs/Channel 11
//     Task_P1 Inputs/IO.I203[12] <-> I203 (GSIO-A-16DIN)/Digital Inputs/Channel 12
//     Task_P1 Inputs/IO.I203[13] <-> I203 (GSIO-A-16DIN)/Digital Inputs/Channel 13
//     Task_P1 Inputs/IO.I203[14] <-> I203 (GSIO-A-16DIN)/Digital Inputs/Channel 14
//     Task_P1 Inputs/IO.I203[15] <-> I203 (GSIO-A-16DIN)/Digital Inputs/Channel 15
//     Task_P1 Inputs/IO.I203[16] <-> I203 (GSIO-A-16DIN)/Digital Inputs/Channel 16
//     Task_P1 Inputs/IO.I203[1] <-> I203 (GSIO-A-16DIN)/Digital Inputs/Channel 1
//     Task_P1 Inputs/IO.I203[2] <-> I203 (GSIO-A-16DIN)/Digital Inputs/Channel 2
//     Task_P1 Inputs/IO.I203[3] <-> I203 (GSIO-A-16DIN)/Digital Inputs/Channel 3
//     Task_P1 Inputs/IO.I203[4] <-> I203 (GSIO-A-16DIN)/Digital Inputs/Channel 4
//     Task_P1 Inputs/IO.I203[5] <-> I203 (GSIO-A-16DIN)/Digital Inputs/Channel 5
//     Task_P1 Inputs/IO.I203[6] <-> I203 (GSIO-A-16DIN)/Digital Inputs/Channel 6
//     Task_P1 Inputs/IO.I203[7] <-> I203 (GSIO-A-16DIN)/Digital Inputs/Channel 7
//     Task_P1 Inputs/IO.I203[8] <-> I203 (GSIO-A-16DIN)/Digital Inputs/Channel 8
//     Task_P1 Inputs/IO.I203[9] <-> I203 (GSIO-A-16DIN)/Digital Inputs/Channel 9
//     Task_P1 Inputs/IO.I204[10] <-> I204 (GSIO-A-16DIN)/Digital Inputs/Channel 10
//     Task_P1 Inputs/IO.I204[11] <-> I204 (GSIO-A-16DIN)/Digital Inputs/Channel 11
//     Task_P1 Inputs/IO.I204[12] <-> I204 (GSIO-A-16DIN)/Digital Inputs/Channel 12
//     Task_P1 Inputs/IO.I204[13] <-> I204 (GSIO-A-16DIN)/Digital Inputs/Channel 13
//     Task_P1 Inputs/IO.I204[14] <-> I204 (GSIO-A-16DIN)/Digital Inputs/Channel 14
//     Task_P1 Inputs/IO.I204[15] <-> I204 (GSIO-A-16DIN)/Digital Inputs/Channel 15
//     Task_P1 Inputs/IO.I204[16] <-> I204 (GSIO-A-16DIN)/Digital Inputs/Channel 16
//     Task_P1 Inputs/IO.I204[1] <-> I204 (GSIO-A-16DIN)/Digital Inputs/Channel 1
//     Task_P1 Inputs/IO.I204[2] <-> I204 (GSIO-A-16DIN)/Digital Inputs/Channel 2
//     Task_P1 Inputs/IO.I204[3] <-> I204 (GSIO-A-16DIN)/Digital Inputs/Channel 3
//     Task_P1 Inputs/IO.I204[4] <-> I204 (GSIO-A-16DIN)/Digital Inputs/Channel 4
//     Task_P1 Inputs/IO.I204[5] <-> I204 (GSIO-A-16DIN)/Digital Inputs/Channel 5
//     Task_P1 Inputs/IO.I204[6] <-> I204 (GSIO-A-16DIN)/Digital Inputs/Channel 6
//     Task_P1 Inputs/IO.I204[7] <-> I204 (GSIO-A-16DIN)/Digital Inputs/Channel 7
//     Task_P1 Inputs/IO.I204[8] <-> I204 (GSIO-A-16DIN)/Digital Inputs/Channel 8
//     Task_P1 Inputs/IO.I204[9] <-> I204 (GSIO-A-16DIN)/Digital Inputs/Channel 9
//     Task_P1 Inputs/IO.I205[10] <-> I205 (GSIO-A-16DIN)/Digital Inputs/Channel 10
//     Task_P1 Inputs/IO.I205[11] <-> I205 (GSIO-A-16DIN)/Digital Inputs/Channel 11
//     Task_P1 Inputs/IO.I205[12] <-> I205 (GSIO-A-16DIN)/Digital Inputs/Channel 12
//     Task_P1 Inputs/IO.I205[13] <-> I205 (GSIO-A-16DIN)/Digital Inputs/Channel 13
//     Task_P1 Inputs/IO.I205[14] <-> I205 (GSIO-A-16DIN)/Digital Inputs/Channel 14
//     Task_P1 Inputs/IO.I205[15] <-> I205 (GSIO-A-16DIN)/Digital Inputs/Channel 15
//     Task_P1 Inputs/IO.I205[16] <-> I205 (GSIO-A-16DIN)/Digital Inputs/Channel 16
//     Task_P1 Inputs/IO.I205[1] <-> I205 (GSIO-A-16DIN)/Digital Inputs/Channel 1
//     Task_P1 Inputs/IO.I205[2] <-> I205 (GSIO-A-16DIN)/Digital Inputs/Channel 2
//     Task_P1 Inputs/IO.I205[3] <-> I205 (GSIO-A-16DIN)/Digital Inputs/Channel 3
//     Task_P1 Inputs/IO.I205[4] <-> I205 (GSIO-A-16DIN)/Digital Inputs/Channel 4
//     Task_P1 Inputs/IO.I205[5] <-> I205 (GSIO-A-16DIN)/Digital Inputs/Channel 5
//     Task_P1 Inputs/IO.I205[6] <-> I205 (GSIO-A-16DIN)/Digital Inputs/Channel 6
//     Task_P1 Inputs/IO.I205[7] <-> I205 (GSIO-A-16DIN)/Digital Inputs/Channel 7
//     Task_P1 Inputs/IO.I205[8] <-> I205 (GSIO-A-16DIN)/Digital Inputs/Channel 8
//     Task_P1 Inputs/IO.I205[9] <-> I205 (GSIO-A-16DIN)/Digital Inputs/Channel 9
//     Task_P1 Inputs/IO.I206[10] <-> I206 (GSIO-A-16DIN)/Digital Inputs/Channel 10
//     Task_P1 Inputs/IO.I206[11] <-> I206 (GSIO-A-16DIN)/Digital Inputs/Channel 11
//     Task_P1 Inputs/IO.I206[12] <-> I206 (GSIO-A-16DIN)/Digital Inputs/Channel 12
//     Task_P1 Inputs/IO.I206[13] <-> I206 (GSIO-A-16DIN)/Digital Inputs/Channel 13
//     Task_P1 Inputs/IO.I206[14] <-> I206 (GSIO-A-16DIN)/Digital Inputs/Channel 14
//     Task_P1 Inputs/IO.I206[15] <-> I206 (GSIO-A-16DIN)/Digital Inputs/Channel 15
//     Task_P1 Inputs/IO.I206[16] <-> I206 (GSIO-A-16DIN)/Digital Inputs/Channel 16
//     Task_P1 Inputs/IO.I206[1] <-> I206 (GSIO-A-16DIN)/Digital Inputs/Channel 1
//     Task_P1 Inputs/IO.I206[2] <-> I206 (GSIO-A-16DIN)/Digital Inputs/Channel 2
//     Task_P1 Inputs/IO.I206[3] <-> I206 (GSIO-A-16DIN)/Digital Inputs/Channel 3
//     Task_P1 Inputs/IO.I206[4] <-> I206 (GSIO-A-16DIN)/Digital Inputs/Channel 4
//     Task_P1 Inputs/IO.I206[5] <-> I206 (GSIO-A-16DIN)/Digital Inputs/Channel 5
//     Task_P1 Inputs/IO.I206[6] <-> I206 (GSIO-A-16DIN)/Digital Inputs/Channel 6
//     Task_P1 Inputs/IO.I206[7] <-> I206 (GSIO-A-16DIN)/Digital Inputs/Channel 7
//     Task_P1 Inputs/IO.I206[8] <-> I206 (GSIO-A-16DIN)/Digital Inputs/Channel 8
//     Task_P1 Inputs/IO.I206[9] <-> I206 (GSIO-A-16DIN)/Digital Inputs/Channel 9
//     Task_P1 Inputs/IO.I207[10] <-> I207 (GSIO-A-16DIN)/Digital Inputs/Channel 10
//     Task_P1 Inputs/IO.I207[11] <-> I207 (GSIO-A-16DIN)/Digital Inputs/Channel 11
//     Task_P1 Inputs/IO.I207[12] <-> I207 (GSIO-A-16DIN)/Digital Inputs/Channel 12
//     Task_P1 Inputs/IO.I207[13] <-> I207 (GSIO-A-16DIN)/Digital Inputs/Channel 13
//     Task_P1 Inputs/IO.I207[14] <-> I207 (GSIO-A-16DIN)/Digital Inputs/Channel 14
//     Task_P1 Inputs/IO.I207[15] <-> I207 (GSIO-A-16DIN)/Digital Inputs/Channel 15
//     Task_P1 Inputs/IO.I207[16] <-> I207 (GSIO-A-16DIN)/Digital Inputs/Channel 16
//     Task_P1 Inputs/IO.I207[1] <-> I207 (GSIO-A-16DIN)/Digital Inputs/Channel 1
//     Task_P1 Inputs/IO.I207[2] <-> I207 (GSIO-A-16DIN)/Digital Inputs/Channel 2
//     Task_P1 Inputs/IO.I207[3] <-> I207 (GSIO-A-16DIN)/Digital Inputs/Channel 3
//     Task_P1 Inputs/IO.I207[4] <-> I207 (GSIO-A-16DIN)/Digital Inputs/Channel 4
//     Task_P1 Inputs/IO.I207[5] <-> I207 (GSIO-A-16DIN)/Digital Inputs/Channel 5
//     Task_P1 Inputs/IO.I207[6] <-> I207 (GSIO-A-16DIN)/Digital Inputs/Channel 6
//     Task_P1 Inputs/IO.I207[7] <-> I207 (GSIO-A-16DIN)/Digital Inputs/Channel 7
//     Task_P1 Inputs/IO.I207[8] <-> I207 (GSIO-A-16DIN)/Digital Inputs/Channel 8
//     Task_P1 Inputs/IO.I207[9] <-> I207 (GSIO-A-16DIN)/Digital Inputs/Channel 9
//     Task_P1 Inputs/IO.I208[10] <-> I208 (GSIO-A-16DIN)/Digital Inputs/Channel 10
//     Task_P1 Inputs/IO.I208[11] <-> I208 (GSIO-A-16DIN)/Digital Inputs/Channel 11
//     Task_P1 Inputs/IO.I208[12] <-> I208 (GSIO-A-16DIN)/Digital Inputs/Channel 12
//     Task_P1 Inputs/IO.I208[13] <-> I208 (GSIO-A-16DIN)/Digital Inputs/Channel 13
//     Task_P1 Inputs/IO.I208[14] <-> I208 (GSIO-A-16DIN)/Digital Inputs/Channel 14
//     Task_P1 Inputs/IO.I208[15] <-> I208 (GSIO-A-16DIN)/Digital Inputs/Channel 15
//     Task_P1 Inputs/IO.I208[16] <-> I208 (GSIO-A-16DIN)/Digital Inputs/Channel 16
//     Task_P1 Inputs/IO.I208[1] <-> I208 (GSIO-A-16DIN)/Digital Inputs/Channel 1
//     Task_P1 Inputs/IO.I208[2] <-> I208 (GSIO-A-16DIN)/Digital Inputs/Channel 2
//     Task_P1 Inputs/IO.I208[3] <-> I208 (GSIO-A-16DIN)/Digital Inputs/Channel 3
//     Task_P1 Inputs/IO.I208[4] <-> I208 (GSIO-A-16DIN)/Digital Inputs/Channel 4
//     Task_P1 Inputs/IO.I208[5] <-> I208 (GSIO-A-16DIN)/Digital Inputs/Channel 5
//     Task_P1 Inputs/IO.I208[6] <-> I208 (GSIO-A-16DIN)/Digital Inputs/Channel 6
//     Task_P1 Inputs/IO.I208[7] <-> I208 (GSIO-A-16DIN)/Digital Inputs/Channel 7
//     Task_P1 Inputs/IO.I208[8] <-> I208 (GSIO-A-16DIN)/Digital Inputs/Channel 8
//     Task_P1 Inputs/IO.I208[9] <-> I208 (GSIO-A-16DIN)/Digital Inputs/Channel 9
//     Task_P1 Inputs/IO.I209[10] <-> I209 (GSIO-A-16DIN)/Digital Inputs/Channel 10
//     Task_P1 Inputs/IO.I209[11] <-> I209 (GSIO-A-16DIN)/Digital Inputs/Channel 11
//     Task_P1 Inputs/IO.I209[12] <-> I209 (GSIO-A-16DIN)/Digital Inputs/Channel 12
//     Task_P1 Inputs/IO.I209[13] <-> I209 (GSIO-A-16DIN)/Digital Inputs/Channel 13
//     Task_P1 Inputs/IO.I209[14] <-> I209 (GSIO-A-16DIN)/Digital Inputs/Channel 14
//     Task_P1 Inputs/IO.I209[15] <-> I209 (GSIO-A-16DIN)/Digital Inputs/Channel 15
//     Task_P1 Inputs/IO.I209[16] <-> I209 (GSIO-A-16DIN)/Digital Inputs/Channel 16
//     Task_P1 Inputs/IO.I209[1] <-> I209 (GSIO-A-16DIN)/Digital Inputs/Channel 1
//     Task_P1 Inputs/IO.I209[2] <-> I209 (GSIO-A-16DIN)/Digital Inputs/Channel 2
//     Task_P1 Inputs/IO.I209[3] <-> I209 (GSIO-A-16DIN)/Digital Inputs/Channel 3
//     Task_P1 Inputs/IO.I209[4] <-> I209 (GSIO-A-16DIN)/Digital Inputs/Channel 4
//     Task_P1 Inputs/IO.I209[5] <-> I209 (GSIO-A-16DIN)/Digital Inputs/Channel 5
//     Task_P1 Inputs/IO.I209[6] <-> I209 (GSIO-A-16DIN)/Digital Inputs/Channel 6
//     Task_P1 Inputs/IO.I209[7] <-> I209 (GSIO-A-16DIN)/Digital Inputs/Channel 7
//     Task_P1 Inputs/IO.I209[8] <-> I209 (GSIO-A-16DIN)/Digital Inputs/Channel 8
//     Task_P1 Inputs/IO.I209[9] <-> I209 (GSIO-A-16DIN)/Digital Inputs/Channel 9
//     Task_P1 Outputs/IO.AO201[{0..3}] <-> AO201 (GSIO-A-4AOV)/Analog Outputs/Channel {1..4}  (4 links)
//     Task_P1 Outputs/IO.Q201[10] <-> Q201 (GSIO-A-16DON)/Digital Outputs/Channel 10
//     Task_P1 Outputs/IO.Q201[11] <-> Q201 (GSIO-A-16DON)/Digital Outputs/Channel 11
//     Task_P1 Outputs/IO.Q201[12] <-> Q201 (GSIO-A-16DON)/Digital Outputs/Channel 12
//     Task_P1 Outputs/IO.Q201[13] <-> Q201 (GSIO-A-16DON)/Digital Outputs/Channel 13
//     Task_P1 Outputs/IO.Q201[14] <-> Q201 (GSIO-A-16DON)/Digital Outputs/Channel 14
//     Task_P1 Outputs/IO.Q201[15] <-> Q201 (GSIO-A-16DON)/Digital Outputs/Channel 15
//     Task_P1 Outputs/IO.Q201[16] <-> Q201 (GSIO-A-16DON)/Digital Outputs/Channel 16
//     Task_P1 Outputs/IO.Q201[1] <-> Q201 (GSIO-A-16DON)/Digital Outputs/Channel 1
//     Task_P1 Outputs/IO.Q201[2] <-> Q201 (GSIO-A-16DON)/Digital Outputs/Channel 2
//     Task_P1 Outputs/IO.Q201[3] <-> Q201 (GSIO-A-16DON)/Digital Outputs/Channel 3
//     Task_P1 Outputs/IO.Q201[4] <-> Q201 (GSIO-A-16DON)/Digital Outputs/Channel 4
//     Task_P1 Outputs/IO.Q201[5] <-> Q201 (GSIO-A-16DON)/Digital Outputs/Channel 5
//     Task_P1 Outputs/IO.Q201[6] <-> Q201 (GSIO-A-16DON)/Digital Outputs/Channel 6
//     Task_P1 Outputs/IO.Q201[7] <-> Q201 (GSIO-A-16DON)/Digital Outputs/Channel 7
//     Task_P1 Outputs/IO.Q201[8] <-> Q201 (GSIO-A-16DON)/Digital Outputs/Channel 8
//     Task_P1 Outputs/IO.Q201[9] <-> Q201 (GSIO-A-16DON)/Digital Outputs/Channel 9
//     Task_P1 Outputs/IO.Q202[10] <-> Q202 (GSIO-A-16DON)/Digital Outputs/Channel 10
//     Task_P1 Outputs/IO.Q202[11] <-> Q202 (GSIO-A-16DON)/Digital Outputs/Channel 11
//     Task_P1 Outputs/IO.Q202[12] <-> Q202 (GSIO-A-16DON)/Digital Outputs/Channel 12
//     Task_P1 Outputs/IO.Q202[13] <-> Q202 (GSIO-A-16DON)/Digital Outputs/Channel 13
//     Task_P1 Outputs/IO.Q202[14] <-> Q202 (GSIO-A-16DON)/Digital Outputs/Channel 14
//     Task_P1 Outputs/IO.Q202[15] <-> Q202 (GSIO-A-16DON)/Digital Outputs/Channel 15
//     Task_P1 Outputs/IO.Q202[16] <-> Q202 (GSIO-A-16DON)/Digital Outputs/Channel 16
//     Task_P1 Outputs/IO.Q202[1] <-> Q202 (GSIO-A-16DON)/Digital Outputs/Channel 1
//     Task_P1 Outputs/IO.Q202[2] <-> Q202 (GSIO-A-16DON)/Digital Outputs/Channel 2
//     Task_P1 Outputs/IO.Q202[3] <-> Q202 (GSIO-A-16DON)/Digital Outputs/Channel 3
//     Task_P1 Outputs/IO.Q202[4] <-> Q202 (GSIO-A-16DON)/Digital Outputs/Channel 4
//     Task_P1 Outputs/IO.Q202[5] <-> Q202 (GSIO-A-16DON)/Digital Outputs/Channel 5
//     Task_P1 Outputs/IO.Q202[6] <-> Q202 (GSIO-A-16DON)/Digital Outputs/Channel 6
//     Task_P1 Outputs/IO.Q202[7] <-> Q202 (GSIO-A-16DON)/Digital Outputs/Channel 7
//     Task_P1 Outputs/IO.Q202[8] <-> Q202 (GSIO-A-16DON)/Digital Outputs/Channel 8
//     Task_P1 Outputs/IO.Q202[9] <-> Q202 (GSIO-A-16DON)/Digital Outputs/Channel 9
//     Task_P1 Outputs/IO.Q203[10] <-> Q203 (GSIO-A-16DON)/Digital Outputs/Channel 10
//     Task_P1 Outputs/IO.Q203[11] <-> Q203 (GSIO-A-16DON)/Digital Outputs/Channel 11
//     Task_P1 Outputs/IO.Q203[12] <-> Q203 (GSIO-A-16DON)/Digital Outputs/Channel 12
//     Task_P1 Outputs/IO.Q203[13] <-> Q203 (GSIO-A-16DON)/Digital Outputs/Channel 13
//     Task_P1 Outputs/IO.Q203[14] <-> Q203 (GSIO-A-16DON)/Digital Outputs/Channel 14
//     Task_P1 Outputs/IO.Q203[15] <-> Q203 (GSIO-A-16DON)/Digital Outputs/Channel 15
//     Task_P1 Outputs/IO.Q203[16] <-> Q203 (GSIO-A-16DON)/Digital Outputs/Channel 16
//     Task_P1 Outputs/IO.Q203[1] <-> Q203 (GSIO-A-16DON)/Digital Outputs/Channel 1
//     Task_P1 Outputs/IO.Q203[2] <-> Q203 (GSIO-A-16DON)/Digital Outputs/Channel 2
//     Task_P1 Outputs/IO.Q203[3] <-> Q203 (GSIO-A-16DON)/Digital Outputs/Channel 3
//     Task_P1 Outputs/IO.Q203[4] <-> Q203 (GSIO-A-16DON)/Digital Outputs/Channel 4
//     Task_P1 Outputs/IO.Q203[5] <-> Q203 (GSIO-A-16DON)/Digital Outputs/Channel 5
//     Task_P1 Outputs/IO.Q203[6] <-> Q203 (GSIO-A-16DON)/Digital Outputs/Channel 6
//     Task_P1 Outputs/IO.Q203[7] <-> Q203 (GSIO-A-16DON)/Digital Outputs/Channel 7
//     Task_P1 Outputs/IO.Q203[8] <-> Q203 (GSIO-A-16DON)/Digital Outputs/Channel 8
//     Task_P1 Outputs/IO.Q203[9] <-> Q203 (GSIO-A-16DON)/Digital Outputs/Channel 9
//     Task_P1 Outputs/IO.Q204[10] <-> Q204 (GSIO-A-16DON)/Digital Outputs/Channel 10
//     Task_P1 Outputs/IO.Q204[11] <-> Q204 (GSIO-A-16DON)/Digital Outputs/Channel 11
//     Task_P1 Outputs/IO.Q204[12] <-> Q204 (GSIO-A-16DON)/Digital Outputs/Channel 12
//     Task_P1 Outputs/IO.Q204[13] <-> Q204 (GSIO-A-16DON)/Digital Outputs/Channel 13
//     Task_P1 Outputs/IO.Q204[14] <-> Q204 (GSIO-A-16DON)/Digital Outputs/Channel 14
//     Task_P1 Outputs/IO.Q204[15] <-> Q204 (GSIO-A-16DON)/Digital Outputs/Channel 15
//     Task_P1 Outputs/IO.Q204[16] <-> Q204 (GSIO-A-16DON)/Digital Outputs/Channel 16
//     Task_P1 Outputs/IO.Q204[1] <-> Q204 (GSIO-A-16DON)/Digital Outputs/Channel 1
//     Task_P1 Outputs/IO.Q204[2] <-> Q204 (GSIO-A-16DON)/Digital Outputs/Channel 2
//     Task_P1 Outputs/IO.Q204[3] <-> Q204 (GSIO-A-16DON)/Digital Outputs/Channel 3
//     Task_P1 Outputs/IO.Q204[4] <-> Q204 (GSIO-A-16DON)/Digital Outputs/Channel 4
//     Task_P1 Outputs/IO.Q204[5] <-> Q204 (GSIO-A-16DON)/Digital Outputs/Channel 5
//     Task_P1 Outputs/IO.Q204[6] <-> Q204 (GSIO-A-16DON)/Digital Outputs/Channel 6
//     Task_P1 Outputs/IO.Q204[7] <-> Q204 (GSIO-A-16DON)/Digital Outputs/Channel 7
//     Task_P1 Outputs/IO.Q204[8] <-> Q204 (GSIO-A-16DON)/Digital Outputs/Channel 8
//     Task_P1 Outputs/IO.Q204[9] <-> Q204 (GSIO-A-16DON)/Digital Outputs/Channel 9
//     Task_P1 Outputs/IO.Q205[10] <-> Q205 (GSIO-A-16DON)/Digital Outputs/Channel 10
//     Task_P1 Outputs/IO.Q205[11] <-> Q205 (GSIO-A-16DON)/Digital Outputs/Channel 11
//     Task_P1 Outputs/IO.Q205[12] <-> Q205 (GSIO-A-16DON)/Digital Outputs/Channel 12
//     Task_P1 Outputs/IO.Q205[13] <-> Q205 (GSIO-A-16DON)/Digital Outputs/Channel 13
//     Task_P1 Outputs/IO.Q205[14] <-> Q205 (GSIO-A-16DON)/Digital Outputs/Channel 14
//     Task_P1 Outputs/IO.Q205[15] <-> Q205 (GSIO-A-16DON)/Digital Outputs/Channel 15
//     Task_P1 Outputs/IO.Q205[16] <-> Q205 (GSIO-A-16DON)/Digital Outputs/Channel 16
//     Task_P1 Outputs/IO.Q205[1] <-> Q205 (GSIO-A-16DON)/Digital Outputs/Channel 1
//     Task_P1 Outputs/IO.Q205[2] <-> Q205 (GSIO-A-16DON)/Digital Outputs/Channel 2
//     Task_P1 Outputs/IO.Q205[3] <-> Q205 (GSIO-A-16DON)/Digital Outputs/Channel 3
//     Task_P1 Outputs/IO.Q205[4] <-> Q205 (GSIO-A-16DON)/Digital Outputs/Channel 4
//     Task_P1 Outputs/IO.Q205[5] <-> Q205 (GSIO-A-16DON)/Digital Outputs/Channel 5
//     Task_P1 Outputs/IO.Q205[6] <-> Q205 (GSIO-A-16DON)/Digital Outputs/Channel 6
//     Task_P1 Outputs/IO.Q205[7] <-> Q205 (GSIO-A-16DON)/Digital Outputs/Channel 7
//     Task_P1 Outputs/IO.Q205[8] <-> Q205 (GSIO-A-16DON)/Digital Outputs/Channel 8
//     Task_P1 Outputs/IO.Q205[9] <-> Q205 (GSIO-A-16DON)/Digital Outputs/Channel 9
//     Task_P1 Outputs/IO.Q206[10] <-> Q206 (GSIO-A-16DON)/Digital Outputs/Channel 10
//     Task_P1 Outputs/IO.Q206[11] <-> Q206 (GSIO-A-16DON)/Digital Outputs/Channel 11
//     Task_P1 Outputs/IO.Q206[12] <-> Q206 (GSIO-A-16DON)/Digital Outputs/Channel 12
//     Task_P1 Outputs/IO.Q206[13] <-> Q206 (GSIO-A-16DON)/Digital Outputs/Channel 13
//     Task_P1 Outputs/IO.Q206[14] <-> Q206 (GSIO-A-16DON)/Digital Outputs/Channel 14
//     Task_P1 Outputs/IO.Q206[15] <-> Q206 (GSIO-A-16DON)/Digital Outputs/Channel 15
//     Task_P1 Outputs/IO.Q206[16] <-> Q206 (GSIO-A-16DON)/Digital Outputs/Channel 16
//     Task_P1 Outputs/IO.Q206[1] <-> Q206 (GSIO-A-16DON)/Digital Outputs/Channel 1
//     Task_P1 Outputs/IO.Q206[2] <-> Q206 (GSIO-A-16DON)/Digital Outputs/Channel 2
//     Task_P1 Outputs/IO.Q206[3] <-> Q206 (GSIO-A-16DON)/Digital Outputs/Channel 3
//     Task_P1 Outputs/IO.Q206[4] <-> Q206 (GSIO-A-16DON)/Digital Outputs/Channel 4
//     Task_P1 Outputs/IO.Q206[5] <-> Q206 (GSIO-A-16DON)/Digital Outputs/Channel 5
//     Task_P1 Outputs/IO.Q206[6] <-> Q206 (GSIO-A-16DON)/Digital Outputs/Channel 6
//     Task_P1 Outputs/IO.Q206[7] <-> Q206 (GSIO-A-16DON)/Digital Outputs/Channel 7
//     Task_P1 Outputs/IO.Q206[8] <-> Q206 (GSIO-A-16DON)/Digital Outputs/Channel 8
//     Task_P1 Outputs/IO.Q206[9] <-> Q206 (GSIO-A-16DON)/Digital Outputs/Channel 9
//     Task_P1 Outputs/IO.Q207[10] <-> Q207 (GSIO-A-16DON)/Digital Outputs/Channel 10
//     Task_P1 Outputs/IO.Q207[11] <-> Q207 (GSIO-A-16DON)/Digital Outputs/Channel 11
//     Task_P1 Outputs/IO.Q207[12] <-> Q207 (GSIO-A-16DON)/Digital Outputs/Channel 12
//     Task_P1 Outputs/IO.Q207[13] <-> Q207 (GSIO-A-16DON)/Digital Outputs/Channel 13
//     Task_P1 Outputs/IO.Q207[14] <-> Q207 (GSIO-A-16DON)/Digital Outputs/Channel 14
//     Task_P1 Outputs/IO.Q207[15] <-> Q207 (GSIO-A-16DON)/Digital Outputs/Channel 15
//     Task_P1 Outputs/IO.Q207[16] <-> Q207 (GSIO-A-16DON)/Digital Outputs/Channel 16
//     Task_P1 Outputs/IO.Q207[1] <-> Q207 (GSIO-A-16DON)/Digital Outputs/Channel 1
//     Task_P1 Outputs/IO.Q207[2] <-> Q207 (GSIO-A-16DON)/Digital Outputs/Channel 2
//     Task_P1 Outputs/IO.Q207[3] <-> Q207 (GSIO-A-16DON)/Digital Outputs/Channel 3
//     Task_P1 Outputs/IO.Q207[4] <-> Q207 (GSIO-A-16DON)/Digital Outputs/Channel 4
//     Task_P1 Outputs/IO.Q207[5] <-> Q207 (GSIO-A-16DON)/Digital Outputs/Channel 5
//     Task_P1 Outputs/IO.Q207[6] <-> Q207 (GSIO-A-16DON)/Digital Outputs/Channel 6
//     Task_P1 Outputs/IO.Q207[7] <-> Q207 (GSIO-A-16DON)/Digital Outputs/Channel 7
//     Task_P1 Outputs/IO.Q207[8] <-> Q207 (GSIO-A-16DON)/Digital Outputs/Channel 8
//     Task_P1 Outputs/IO.Q207[9] <-> Q207 (GSIO-A-16DON)/Digital Outputs/Channel 9
//     Task_P1 Outputs/IO.Q208[10] <-> Q208 (GSIO-A-16DON)/Digital Outputs/Channel 10
//     Task_P1 Outputs/IO.Q208[11] <-> Q208 (GSIO-A-16DON)/Digital Outputs/Channel 11
//     Task_P1 Outputs/IO.Q208[12] <-> Q208 (GSIO-A-16DON)/Digital Outputs/Channel 12
//     Task_P1 Outputs/IO.Q208[13] <-> Q208 (GSIO-A-16DON)/Digital Outputs/Channel 13
//     Task_P1 Outputs/IO.Q208[14] <-> Q208 (GSIO-A-16DON)/Digital Outputs/Channel 14
//     Task_P1 Outputs/IO.Q208[15] <-> Q208 (GSIO-A-16DON)/Digital Outputs/Channel 15
//     Task_P1 Outputs/IO.Q208[16] <-> Q208 (GSIO-A-16DON)/Digital Outputs/Channel 16
//     Task_P1 Outputs/IO.Q208[1] <-> Q208 (GSIO-A-16DON)/Digital Outputs/Channel 1
//     Task_P1 Outputs/IO.Q208[2] <-> Q208 (GSIO-A-16DON)/Digital Outputs/Channel 2
//     Task_P1 Outputs/IO.Q208[3] <-> Q208 (GSIO-A-16DON)/Digital Outputs/Channel 3
//     Task_P1 Outputs/IO.Q208[4] <-> Q208 (GSIO-A-16DON)/Digital Outputs/Channel 4
//     Task_P1 Outputs/IO.Q208[5] <-> Q208 (GSIO-A-16DON)/Digital Outputs/Channel 5
//     Task_P1 Outputs/IO.Q208[6] <-> Q208 (GSIO-A-16DON)/Digital Outputs/Channel 6
//     Task_P1 Outputs/IO.Q208[7] <-> Q208 (GSIO-A-16DON)/Digital Outputs/Channel 7
//     Task_P1 Outputs/IO.Q208[8] <-> Q208 (GSIO-A-16DON)/Digital Outputs/Channel 8
//     Task_P1 Outputs/IO.Q208[9] <-> Q208 (GSIO-A-16DON)/Digital Outputs/Channel 9
//     Task_P1 Outputs/IO.Q209[10] <-> Q209 (GSIO-A-16DON)/Digital Outputs/Channel 10
//     Task_P1 Outputs/IO.Q209[11] <-> Q209 (GSIO-A-16DON)/Digital Outputs/Channel 11
//     Task_P1 Outputs/IO.Q209[12] <-> Q209 (GSIO-A-16DON)/Digital Outputs/Channel 12
//     Task_P1 Outputs/IO.Q209[13] <-> Q209 (GSIO-A-16DON)/Digital Outputs/Channel 13
//     Task_P1 Outputs/IO.Q209[14] <-> Q209 (GSIO-A-16DON)/Digital Outputs/Channel 14
//     Task_P1 Outputs/IO.Q209[15] <-> Q209 (GSIO-A-16DON)/Digital Outputs/Channel 15
//     Task_P1 Outputs/IO.Q209[16] <-> Q209 (GSIO-A-16DON)/Digital Outputs/Channel 16
//     Task_P1 Outputs/IO.Q209[1] <-> Q209 (GSIO-A-16DON)/Digital Outputs/Channel 1
//     Task_P1 Outputs/IO.Q209[2] <-> Q209 (GSIO-A-16DON)/Digital Outputs/Channel 2
//     Task_P1 Outputs/IO.Q209[3] <-> Q209 (GSIO-A-16DON)/Digital Outputs/Channel 3
//     Task_P1 Outputs/IO.Q209[4] <-> Q209 (GSIO-A-16DON)/Digital Outputs/Channel 4
//     Task_P1 Outputs/IO.Q209[5] <-> Q209 (GSIO-A-16DON)/Digital Outputs/Channel 5
//     Task_P1 Outputs/IO.Q209[6] <-> Q209 (GSIO-A-16DON)/Digital Outputs/Channel 6
//     Task_P1 Outputs/IO.Q209[7] <-> Q209 (GSIO-A-16DON)/Digital Outputs/Channel 7
//     Task_P1 Outputs/IO.Q209[8] <-> Q209 (GSIO-A-16DON)/Digital Outputs/Channel 8
//     Task_P1 Outputs/IO.Q209[9] <-> Q209 (GSIO-A-16DON)/Digital Outputs/Channel 9
//   MQPLC/MQPLC Instance <-> Device 3 (EtherCAT)/P2M1正极送料分段皮带1[20(模切)] (InoSV660N)
//     Task_P1 Inputs/GMotion.arrAxisCtrl[20].Io.ErrorCode <-> Inputs/Error code
//     Task_P1 Inputs/GMotion.iActTorque_M[20] <-> Inputs/Torque actual value
//   MQPLC/MQPLC Instance <-> Device 3 (EtherCAT)/P2M1负极送料分段皮带1[44（模切）] (InoSV660N)
//     Task_P1 Inputs/GMotion.arrAxisCtrl[44].Io.ErrorCode <-> Inputs/Error code
//     Task_P1 Inputs/GMotion.iActTorque_M[44] <-> Inputs/Torque actual value
//   MQPLC/MQPLC Instance <-> NC-Task 1 SAF/Axes/Axis001_1 P1An_UnWind_L
//     Task_P1 Inputs/GMotion.arrAxis[1].NcToPlc <-> Outputs/ToPlc
//     Task_P1 Outputs/GMotion.arrAxis[1].PlcToNc <-> Inputs/FromPlc
//   MQPLC/MQPLC Instance <-> NC-Task 1 SAF/Axes/Axis002_2 P1An_UnWind_R
//     Task_P1 Inputs/GMotion.arrAxis[2].NcToPlc <-> Outputs/ToPlc
//     Task_P1 Outputs/GMotion.arrAxis[2].PlcToNc <-> Inputs/FromPlc
//   MQPLC/MQPLC Instance <-> NC-Task 1 SAF/Axes/Axis003_3 P1An_PoleTension
//     Task_P1 Inputs/GMotion.arrAxis[3].NcToPlc <-> Outputs/ToPlc
//     Task_P1 Outputs/GMotion.arrAxis[3].PlcToNc <-> Inputs/FromPlc
//   MQPLC/MQPLC Instance <-> NC-Task 1 SAF/Axes/Axis004_4 P1An_DriverAux
//     Task_P1 Inputs/GMotion.arrAxis[4].NcToPlc <-> Outputs/ToPlc
//     Task_P1 Outputs/GMotion.arrAxis[4].PlcToNc <-> Inputs/FromPlc
//   MQPLC/MQPLC Instance <-> NC-Task 1 SAF/Axes/Axis005_5 P1An_BuffeLine
//     Task_P1 Inputs/GMotion.arrAxis[5].NcToPlc <-> Outputs/ToPlc
//     Task_P1 Outputs/GMotion.arrAxis[5].PlcToNc <-> Inputs/FromPlc
//   MQPLC/MQPLC Instance <-> NC-Task 1 SAF/Axes/Axis006_6 P1An_Mould
//     Task_P1 Inputs/GMotion.arrAxis[6].NcToPlc <-> Outputs/ToPlc
//     Task_P1 Outputs/GMotion.arrAxis[6].PlcToNc <-> Inputs/FromPlc
//   MQPLC/MQPLC Instance <-> NC-Task 1 SAF/Axes/Axis007_7 P1An_MouldRectify_X
//     Task_P1 Inputs/GMotion.arrAxis[7].NcToPlc <-> Outputs/ToPlc
//     Task_P1 Outputs/GMotion.arrAxis[7].PlcToNc <-> Inputs/FromPlc
//   MQPLC/MQPLC Instance <-> NC-Task 1 SAF/Axes/Axis008_8 P1An_MouldRectify_Y
//     Task_P1 Inputs/GMotion.arrAxis[8].NcToPlc <-> Outputs/ToPlc
//     Task_P1 Outputs/GMotion.arrAxis[8].PlcToNc <-> Inputs/FromPlc
//   MQPLC/MQPLC Instance <-> NC-Task 1 SAF/Axes/Axis009_9 P1An_DriverDDR
//     Task_P1 Inputs/GMotion.arrAxis[9].NcToPlc <-> Outputs/ToPlc
//     Task_P1 Outputs/GMotion.arrAxis[9].PlcToNc <-> Inputs/FromPlc
//   MQPLC/MQPLC Instance <-> NC-Task 1 SAF/Axes/Axis010_10 P1An_Cuter
//     Task_P1 Inputs/GMotion.arrAxis[10].NcToPlc <-> Outputs/ToPlc
//     Task_P1 Outputs/GMotion.arrAxis[10].PlcToNc <-> Inputs/FromPlc
//   MQPLC/MQPLC Instance <-> NC-Task 1 SAF/Axes/Axis011_11 P1An_CuterDegRectify
//     Task_P1 Inputs/GMotion.arrAxis[11].NcToPlc <-> Outputs/ToPlc
//     Task_P1 Outputs/GMotion.arrAxis[11].PlcToNc <-> Inputs/FromPlc
//   MQPLC/MQPLC Instance <-> NC-Task 1 SAF/Axes/Axis012_12 P1An_CuterBelt
//     Task_P1 Inputs/GMotion.arrAxis[12].NcToPlc <-> Outputs/ToPlc
//     Task_P1 Outputs/GMotion.arrAxis[12].PlcToNc <-> Inputs/FromPlc
//   MQPLC/MQPLC Instance <-> NC-Task 1 SAF/Axes/Axis013_13 P1An_CuterBeltChange
//     Task_P1 Inputs/GMotion.arrAxis[13].NcToPlc <-> Outputs/ToPlc
//     Task_P1 Outputs/GMotion.arrAxis[13].PlcToNc <-> Inputs/FromPlc
//   MQPLC/MQPLC Instance <-> NC-Task 1 SAF/Axes/Axis014_14 P1An_CCDPressPush
//     Task_P1 Inputs/GMotion.arrAxis[14].NcToPlc <-> Outputs/ToPlc
//     Task_P1 Outputs/GMotion.arrAxis[14].PlcToNc <-> Inputs/FromPlc
//   MQPLC/MQPLC Instance <-> NC-Task 1 SAF/Axes/Axis015_15 P1An_NGPushReverseBelt
//     Task_P1 Inputs/GMotion.arrAxis[15].NcToPlc <-> Outputs/ToPlc
//     Task_P1 Outputs/GMotion.arrAxis[15].PlcToNc <-> Inputs/FromPlc
//   MQPLC/MQPLC Instance <-> NC-Task 1 SAF/Axes/Axis016_16 P1An_NGPush1
//     Task_P1 Inputs/GMotion.arrAxis[16].NcToPlc <-> Outputs/ToPlc
//     Task_P1 Outputs/GMotion.arrAxis[16].PlcToNc <-> Inputs/FromPlc
//   MQPLC/MQPLC Instance <-> NC-Task 1 SAF/Axes/Axis017_17 P1An_NGPush2
//     Task_P1 Inputs/GMotion.arrAxis[17].NcToPlc <-> Outputs/ToPlc
//     Task_P1 Outputs/GMotion.arrAxis[17].PlcToNc <-> Inputs/FromPlc
//   MQPLC/MQPLC Instance <-> NC-Task 1 SAF/Axes/Axis018_18 P1An_DedustBelt
//     Task_P1 Inputs/GMotion.arrAxis[18].NcToPlc <-> Outputs/ToPlc
//     Task_P1 Outputs/GMotion.arrAxis[18].PlcToNc <-> Inputs/FromPlc
//   MQPLC/MQPLC Instance <-> NC-Task 1 SAF/Axes/Axis019_19 P1An_DedustReverseBelt
//     Task_P1 Inputs/GMotion.arrAxis[19].NcToPlc <-> Outputs/ToPlc
//     Task_P1 Outputs/GMotion.arrAxis[19].PlcToNc <-> Inputs/FromPlc
//   MQPLC/MQPLC Instance <-> NC-Task 1 SAF/Axes/Axis020_20 P1An_SubBelt1
//     Task_P1 Inputs/GMotion.arrAxis[20].NcToPlc <-> Outputs/ToPlc
//     Task_P1 Outputs/GMotion.arrAxis[20].PlcToNc <-> Inputs/FromPlc
//   MQPLC/MQPLC Instance <-> NC-Task 1 SAF/Axes/Axis021_21 P1An_SubBelt2
//     Task_P1 Inputs/GMotion.arrAxis[21].NcToPlc <-> Outputs/ToPlc
//     Task_P1 Outputs/GMotion.arrAxis[21].PlcToNc <-> Inputs/FromPlc
//   MQPLC/MQPLC Instance <-> NC-Task 1 SAF/Axes/Axis022_22 P1An_SubBelt3
//     Task_P1 Inputs/GMotion.arrAxis[22].NcToPlc <-> Outputs/ToPlc
//     Task_P1 Outputs/GMotion.arrAxis[22].PlcToNc <-> Inputs/FromPlc
//   MQPLC/MQPLC Instance <-> NC-Task 1 SAF/Axes/Axis023_23 P1An_Ready1
//     Task_P1 Inputs/GMotion.arrAxis[23].NcToPlc <-> Outputs/ToPlc
//     Task_P1 Outputs/GMotion.arrAxis[23].PlcToNc <-> Inputs/FromPlc
//   MQPLC/MQPLC Instance <-> NC-Task 1 SAF/Axes/Axis024_24 P1An_Ready2
//     Task_P1 Inputs/GMotion.arrAxis[24].NcToPlc <-> Outputs/ToPlc
//     Task_P1 Outputs/GMotion.arrAxis[24].PlcToNc <-> Inputs/FromPlc
//   MQPLC/MQPLC Instance <-> NC-Task 1 SAF/Axes/Axis025_25 P1Ca_UnWind_L
//     Task_P1 Inputs/GMotion.arrAxis[25].NcToPlc <-> Outputs/ToPlc
//     Task_P1 Outputs/GMotion.arrAxis[25].PlcToNc <-> Inputs/FromPlc
//   MQPLC/MQPLC Instance <-> NC-Task 1 SAF/Axes/Axis026_26 P1Ca_UnWind_R
//     Task_P1 Inputs/GMotion.arrAxis[26].NcToPlc <-> Outputs/ToPlc
//     Task_P1 Outputs/GMotion.arrAxis[26].PlcToNc <-> Inputs/FromPlc
//   MQPLC/MQPLC Instance <-> NC-Task 1 SAF/Axes/Axis027_27 P1Ca_PoleTension
//     Task_P1 Inputs/GMotion.arrAxis[27].NcToPlc <-> Outputs/ToPlc
//     Task_P1 Outputs/GMotion.arrAxis[27].PlcToNc <-> Inputs/FromPlc
//   MQPLC/MQPLC Instance <-> NC-Task 1 SAF/Axes/Axis028_28 P1Ca_DriverAux
//     Task_P1 Inputs/GMotion.arrAxis[28].NcToPlc <-> Outputs/ToPlc
//     Task_P1 Outputs/GMotion.arrAxis[28].PlcToNc <-> Inputs/FromPlc
//   MQPLC/MQPLC Instance <-> NC-Task 1 SAF/Axes/Axis029_29 P1Ca_BuffeLine
//     Task_P1 Inputs/GMotion.arrAxis[29].NcToPlc <-> Outputs/ToPlc
//     Task_P1 Outputs/GMotion.arrAxis[29].PlcToNc <-> Inputs/FromPlc
//   MQPLC/MQPLC Instance <-> NC-Task 1 SAF/Axes/Axis030_30 P1Ca_Mould
//     Task_P1 Inputs/GMotion.arrAxis[30].NcToPlc <-> Outputs/ToPlc
//     Task_P1 Outputs/GMotion.arrAxis[30].PlcToNc <-> Inputs/FromPlc
//   MQPLC/MQPLC Instance <-> NC-Task 1 SAF/Axes/Axis031_31 P1Ca_MouldRectify_X
//     Task_P1 Inputs/GMotion.arrAxis[31].NcToPlc <-> Outputs/ToPlc
//     Task_P1 Outputs/GMotion.arrAxis[31].PlcToNc <-> Inputs/FromPlc
//   MQPLC/MQPLC Instance <-> NC-Task 1 SAF/Axes/Axis032_32 P1Ca_MouldRectify_Y
//     Task_P1 Inputs/GMotion.arrAxis[32].NcToPlc <-> Outputs/ToPlc
//     Task_P1 Outputs/GMotion.arrAxis[32].PlcToNc <-> Inputs/FromPlc
//   MQPLC/MQPLC Instance <-> NC-Task 1 SAF/Axes/Axis033_33 P1Ca_DriverDDR
//     Task_P1 Inputs/GMotion.arrAxis[33].NcToPlc <-> Outputs/ToPlc
//     Task_P1 Outputs/GMotion.arrAxis[33].PlcToNc <-> Inputs/FromPlc
//   MQPLC/MQPLC Instance <-> NC-Task 1 SAF/Axes/Axis034_34 P1Ca_Cuter
//     Task_P1 Inputs/GMotion.arrAxis[34].NcToPlc <-> Outputs/ToPlc
//     Task_P1 Outputs/GMotion.arrAxis[34].PlcToNc <-> Inputs/FromPlc
//   MQPLC/MQPLC Instance <-> NC-Task 1 SAF/Axes/Axis035_35 P1Ca_CuterDegRectify
//     Task_P1 Inputs/GMotion.arrAxis[35].NcToPlc <-> Outputs/ToPlc
//     Task_P1 Outputs/GMotion.arrAxis[35].PlcToNc <-> Inputs/FromPlc
//   MQPLC/MQPLC Instance <-> NC-Task 1 SAF/Axes/Axis036_36 P1Ca_CuterBelt
//     Task_P1 Inputs/GMotion.arrAxis[36].NcToPlc <-> Outputs/ToPlc
//     Task_P1 Outputs/GMotion.arrAxis[36].PlcToNc <-> Inputs/FromPlc
//   MQPLC/MQPLC Instance <-> NC-Task 1 SAF/Axes/Axis037_37 P1Ca_CuterBeltChange
//     Task_P1 Inputs/GMotion.arrAxis[37].NcToPlc <-> Outputs/ToPlc
//     Task_P1 Outputs/GMotion.arrAxis[37].PlcToNc <-> Inputs/FromPlc
//   MQPLC/MQPLC Instance <-> NC-Task 1 SAF/Axes/Axis038_38 P1Ca_CCDPressPush
//     Task_P1 Inputs/GMotion.arrAxis[38].NcToPlc <-> Outputs/ToPlc
//     Task_P1 Outputs/GMotion.arrAxis[38].PlcToNc <-> Inputs/FromPlc
//   MQPLC/MQPLC Instance <-> NC-Task 1 SAF/Axes/Axis039_39 P1Ca_NGPushReverseBelt
//     Task_P1 Inputs/GMotion.arrAxis[39].NcToPlc <-> Outputs/ToPlc
//     Task_P1 Outputs/GMotion.arrAxis[39].PlcToNc <-> Inputs/FromPlc
//   MQPLC/MQPLC Instance <-> NC-Task 1 SAF/Axes/Axis040_40 P1Ca_NGPush1
//     Task_P1 Inputs/GMotion.arrAxis[40].NcToPlc <-> Outputs/ToPlc
//     Task_P1 Outputs/GMotion.arrAxis[40].PlcToNc <-> Inputs/FromPlc
//   MQPLC/MQPLC Instance <-> NC-Task 1 SAF/Axes/Axis041_41 P1Ca_NGPush2
//     Task_P1 Inputs/GMotion.arrAxis[41].NcToPlc <-> Outputs/ToPlc
//     Task_P1 Outputs/GMotion.arrAxis[41].PlcToNc <-> Inputs/FromPlc
//   MQPLC/MQPLC Instance <-> NC-Task 1 SAF/Axes/Axis042_42 P1Ca_DedustBelt
//     Task_P1 Inputs/GMotion.arrAxis[42].NcToPlc <-> Outputs/ToPlc
//     Task_P1 Outputs/GMotion.arrAxis[42].PlcToNc <-> Inputs/FromPlc
//   MQPLC/MQPLC Instance <-> NC-Task 1 SAF/Axes/Axis043_43 P1Ca_DedustReverseBelt
//     Task_P1 Inputs/GMotion.arrAxis[43].NcToPlc <-> Outputs/ToPlc
//     Task_P1 Outputs/GMotion.arrAxis[43].PlcToNc <-> Inputs/FromPlc
//   MQPLC/MQPLC Instance <-> NC-Task 1 SAF/Axes/Axis044_44 P1Ca_SubBelt1
//     Task_P1 Inputs/GMotion.arrAxis[44].NcToPlc <-> Outputs/ToPlc
//     Task_P1 Outputs/GMotion.arrAxis[44].PlcToNc <-> Inputs/FromPlc
//   MQPLC/MQPLC Instance <-> NC-Task 1 SAF/Axes/Axis045_45 P1Ca_SubBelt2
//     Task_P1 Inputs/GMotion.arrAxis[45].NcToPlc <-> Outputs/ToPlc
//     Task_P1 Outputs/GMotion.arrAxis[45].PlcToNc <-> Inputs/FromPlc
//   MQPLC/MQPLC Instance <-> NC-Task 1 SAF/Axes/Axis046_46 P1Ca_SubBelt3
//     Task_P1 Inputs/GMotion.arrAxis[46].NcToPlc <-> Outputs/ToPlc
//     Task_P1 Outputs/GMotion.arrAxis[46].PlcToNc <-> Inputs/FromPlc
//   MQPLC/MQPLC Instance <-> NC-Task 1 SAF/Axes/Axis047_47 P1Ca_Ready1
//     Task_P1 Inputs/GMotion.arrAxis[47].NcToPlc <-> Outputs/ToPlc
//     Task_P1 Outputs/GMotion.arrAxis[47].PlcToNc <-> Inputs/FromPlc
//   MQPLC/MQPLC Instance <-> NC-Task 1 SAF/Axes/Axis048_48 P1Ca_Ready2
//     Task_P1 Inputs/GMotion.arrAxis[48].NcToPlc <-> Outputs/ToPlc
//     Task_P1 Outputs/GMotion.arrAxis[48].PlcToNc <-> Inputs/FromPlc
//   MQPLC/MQPLC Instance <-> NC-Task 1 SAF/Axes/Axis210_50 P1_VirTimeWind
//     Task_P1 Inputs/GMotion.arrAxis[50].NcToPlc <-> Outputs/ToPlc
//     Task_P1 Outputs/GMotion.arrAxis[50].PlcToNc <-> Inputs/FromPlc
//   MQPLC/MQPLC Instance <-> NC-Task 1 SAF/Axes/Axis211_51 P1An_VirMain
//     Task_P1 Inputs/GMotion.arrAxis[51].NcToPlc <-> Outputs/ToPlc
//     Task_P1 Outputs/GMotion.arrAxis[51].PlcToNc <-> Inputs/FromPlc
//   MQPLC/MQPLC Instance <-> NC-Task 1 SAF/Axes/Axis212_52 P1An_VirDriver
//     Task_P1 Inputs/GMotion.arrAxis[52].NcToPlc <-> Outputs/ToPlc
//     Task_P1 Outputs/GMotion.arrAxis[52].PlcToNc <-> Inputs/FromPlc
//   MQPLC/MQPLC Instance <-> NC-Task 1 SAF/Axes/Axis213_53 P1An_VirBelt
//     Task_P1 Inputs/GMotion.arrAxis[53].NcToPlc <-> Outputs/ToPlc
//     Task_P1 Outputs/GMotion.arrAxis[53].PlcToNc <-> Inputs/FromPlc
//   MQPLC/MQPLC Instance <-> NC-Task 1 SAF/Axes/Axis214_56 P1Ca_VirMain
//     Task_P1 Inputs/GMotion.arrAxis[56].NcToPlc <-> Outputs/ToPlc
//     Task_P1 Outputs/GMotion.arrAxis[56].PlcToNc <-> Inputs/FromPlc
//   MQPLC/MQPLC Instance <-> NC-Task 1 SAF/Axes/Axis215_57 P1Ca_VirDriver
//     Task_P1 Inputs/GMotion.arrAxis[57].NcToPlc <-> Outputs/ToPlc
//     Task_P1 Outputs/GMotion.arrAxis[57].PlcToNc <-> Inputs/FromPlc
//   MQPLC/MQPLC Instance <-> NC-Task 1 SAF/Axes/Axis216_58 P1Ca_VirBelt
//     Task_P1 Inputs/GMotion.arrAxis[58].NcToPlc <-> Outputs/ToPlc
//     Task_P1 Outputs/GMotion.arrAxis[58].PlcToNc <-> Inputs/FromPlc

CONFIGURATION DPPLC
    RESOURCE PLC ON TwinCAT3
        TASK Task_P2M1(INTERVAL := T#2ms, PRIORITY := 16);
        TASK Task_P2M2(INTERVAL := T#2ms, PRIORITY := 14);
        TASK Task_P2M3(INTERVAL := T#2ms, PRIORITY := 12);
        TASK Task_P2Main(INTERVAL := T#2ms, PRIORITY := 10);
        TASK Task_P3(INTERVAL := T#2ms, PRIORITY := 18);
        PROGRAM P2M1_Auto WITH Task_P2M1 : P2M1_Auto;
        PROGRAM P2M2_Auto WITH Task_P2M2 : P2M2_Auto;
        PROGRAM P2M3_Auto WITH Task_P2M3 : P2M3_Auto;
        PROGRAM MAIN WITH Task_P2Main : MAIN;
        PROGRAM P3MAIN WITH Task_P3 : P3MAIN;
    END_RESOURCE
END_CONFIGURATION

// ---- P2DUTs/01_AxisCO_Ntrol/MC_AxisParameter.TcDUT


TYPE MC_AxisParameter : (
(* PLCopen specific parameters *) (* Index-Group 0x4000 + ID*)
   CommandedPosition := 1,           (* lreal *) (* taken from NcToPlc *)
   SWLimitPos,                       (* lreal *) (* IndexOffset= 16#0001_000E *)
   SWLimitNeg,                       (* lreal *) (* IndexOffset= 16#0001_000D *)
   EnableLimitPos,                   (* bool  *) (* IndexOffset= 16#0001_000C *)
   EnableLimitNeg,                   (* bool  *) (* IndexOffset= 16#0001_000B *)
   EnablePosLagMonitoring,           (* bool  *) (* IndexOffset= 16#0002_0010 *)
   MaxPositionLag,                   (* lreal *) (* IndexOffset= 16#0002_0012 *)
   MaxVelocitySystem,                (* lreal *) (* IndexOffset= 16#0000_0027 *)
   MaxVelocityAppl,                  (* lreal *) (* IndexOffset= 16#0000_0027 *)
   ActualVelocity,                   (* lreal *) (* taken from NcToPlc *)
   CommandedVelocity,                (* lreal *) (* taken from NcToPlc *)
   MaxAccelerationSystem,            (* lreal *) (* IndexOffset= 16#0000_0101 *)
   MaxAccelerationAppl,              (* lreal *) (* IndexOffset= 16#0000_0101 *)
   MaxDecelerationSystem,            (* lreal *) (* IndexOffset= 16#0000_0102 *)
   MaxDecelerationAppl,              (* lreal *) (* IndexOffset= 16#0000_0102 *)
   MaxJerkSystem,                    (* lreal *) (* IndexOffset= 16#0000_0103 *)
   MaxJerkAppl,                      (* lreal *) (* IndexOffset= 16#0000_0103 *)

(* Beckhoff specific parameters *) (* Index-Group 0x4000 + ID*)
   AxisId := 1000,                   (* lreal *) (* IndexOffset= 16#0000_0001 *)
   AxisVeloManSlow,                  (* lreal *) (* IndexOffset= 16#0000_0008 *)
   AxisVeloManFast,                  (* lreal *) (* IndexOffset= 16#0000_0009 *)
   AxisVeloMax,                      (* lreal *) (* IndexOffset= 16#0000_0027 *)
   AxisAcc,                          (* lreal *) (* IndexOffset= 16#0000_0101 *)
   AxisDec,                          (* lreal *) (* IndexOffset= 16#0000_0102 *)
   AxisJerk,                         (* lreal *) (* IndexOffset= 16#0000_0103 *)
   MaxJerk,                          (* lreal *) (* IndexOffset= 16#0000_0103 *)
   AxisMaxVelocity,                  (* lreal *) (* IndexOffset= 16#0000_0027 *)
   AxisRapidTraverseVelocity,        (* lreal *) (* IndexOffset= 16#0000_000A *)
   AxisManualVelocityFast,           (* lreal *) (* IndexOffset= 16#0000_0009 *)
   AxisManualVelocitySlow,           (* lreal *) (* IndexOffset= 16#0000_0008 *)
   AxisCalibrationVelocityForward,   (* lreal *) (* IndexOffset= 16#0000_0006 *)
   AxisCalibrationVelocityBackward,  (* lreal *) (* IndexOffset= 16#0000_0007 *)
   AxisJogIncrementForward,          (* lreal *) (* IndexOffset= 16#0000_0018 *)
   AxisJogIncrementBackward,         (* lreal *) (* IndexOffset= 16#0000_0019 *)
   AxisEnMinSoftPosLimit,            (* bool  *) (* IndexOffset= 16#0001_000B *)
   AxisMinSoftPosLimit,              (* lreal *) (* IndexOffset= 16#0001_000D *)
   AxisEnMaxSoftPosLimit,            (* bool  *) (* IndexOffset= 16#0001_000C *)
   AxisMaxSoftPosLimit,              (* lreal *) (* IndexOffset= 16#0001_000E *)
   AxisEnPositionLagMonitoring,      (* bool  *) (* IndexOffset= 16#0002_0010 *)
   AxisMaxPosLagValue,               (* lreal *) (* IndexOffset= 16#0002_0012 *)
   AxisMaxPosLagFilterTime,          (* lreal *) (* IndexOffset= 16#0002_0013 *)
   AxisEnPositionRangeMonitoring,    (* bool  *) (* IndexOffset= 16#0000_000F *)
   AxisPositionRangeWindow,          (* lreal *) (* IndexOffset= 16#0000_0010 *)
   AxisEnTargetPositionMonitoring,   (* bool  *) (* IndexOffset= 16#0000_0015 *)
   AxisTargetPositionWindow,         (* lreal *) (* IndexOffset= 16#0000_0016 *)
   AxisTargetPositionMonitoringTime, (* lreal *) (* IndexOffset= 16#0000_0017 *)
   AxisEnInTargetTimeout,            (* bool  *) (* IndexOffset= 16#0000_0029 *)
   AxisInTargetTimeout,              (* lreal *) (* IndexOffset= 16#0000_002A *)
   AxisEnMotionMonitoring,           (* bool  *) (* IndexOffset= 16#0000_0011 *)
   AxisMotionMonitoringWindow,       (* lreal *) (* IndexOffset= 16#0000_0028 *)
   AxisMotionMonitoringTime,         (* lreal *) (* IndexOffset= 16#0000_0012 *)
   AxisDelayTimeVeloPosition,        (* lreal *) (* IndexOffset= 16#0000_0104 *)
   AxisEnLoopingDistance,            (* bool  *) (* IndexOffset= 16#0000_0013 *)
   AxisLoopingDistance,              (* lreal *) (* IndexOffset= 16#0000_0014 *)
   AxisEnBacklashCompensation,       (* bool  *) (* IndexOffset= 16#0000_002B *)
   AxisBacklash,                     (* lreal *) (* IndexOffset= 16#0000_002C *)
   AxisEnDataPersistence,            (* bool  *) (* IndexOffset= 16#0000_0030 *)
   AxisRefVeloOnRefOutput,           (* lreal *) (* IndexOffset= 16#0003_0101 *)
   AxisOverrideType,                 (* lreal *) (* IndexOffset= 16#0000_0105 *)
   (* new since 4/2007 *)
   AxisEncoderScalingFactor,         (* lreal *) (* IndexOffset= 16#0001_0006 *)
   AxisEncoderOffset,                (* lreal *) (* IndexOffset= 16#0001_0007 *)
   AxisEncoderDirectionInverse,      (* bool  *) (* IndexOffset= 16#0001_0008 *)
   AxisEncoderMask,                  (* dword *) (* IndexOffset= 16#0001_0015 *)
   AxisEncoderModuloValue,           (* lreal *) (* IndexOffset= 16#0001_0009 *)
   AxisModuloToleranceWindow,        (* lreal *) (* IndexOffset= 16#0001_001B *)
   AxisEnablePosCorrection,          (* bool  *) (* IndexOffset= 16#0001_0016 *)
   AxisPosCorrectionFilterTime,      (* lreal *) (* IndexOffset= 16#0001_0017 *)
   (* new since 1/2010 *)
   AxisUnitInterpretation,           (* lreal *) (* IndexOffset= 16#0000_0026 *)
   AxisMotorDirectionInverse,        (* bool  *) (* IndexOffset= 16#0003_0006 *)
   (* new since 1/2011 *)
   AxisCycleTime,                    (* lreal *) (* IndexOffset= 16#0000_0004 *)
   (* new since 5/2011 *)
   AxisFastStopSignalType,           (* dword *) (* IndexOffset= 16#0000_001E *)
   AxisFastAcc,                      (* lreal *) (* IndexOffset= 16#0000_010A *)
   AxisFastDec,                      (* lreal *) (* IndexOffset= 16#0000_010B *)
   AxisFastJerk,                     (* lreal *) (* IndexOffset= 16#0000_010C *)

(* Beckhoff specific axis status information - READ ONLY *) (* Index-Group 0x4100 + ID*)
   AxisTargetPosition := 2000,       (* lreal *) (* IndexOffset= 16#0000_0013 *)
   AxisRemainingTimeToGo,            (* lreal *) (* IndexOffset= 16#0000_0014 *)
   AxisRemainingDistanceToGo,        (* lreal *) (* IndexOffset= 16#0000_0022, 16#0000_0042 *)

(* Beckhoff specific axis functions *)
   (* read/write gear ratio of a slave *)
   AxisGearRatio := 3000,            (* lreal *) (* read: IndexGroup=0x4100+ID, IdxOffset=16#0000_0022, *)
                   (* write:IndexGroup=0x4200+ID, IdxOffset=16#0000_0042 *) 

(* Beckhoff specific other parameters *)
   (* new since 1/2011 *)
   NcSafCycleTime := 4000,           (* lreal *) (* IndexOffset= 16#0000_0010 *)
   NcSvbCycleTime                    (* lreal *) (* IndexOffset= 16#0000_0012 *)
);
END_TYPE

// ---- P2DUTs/01_AxisCO_Ntrol/ST_Dust_Motor.TcDUT
TYPE ST_Dust_Motor :
STRUCT
	bJog_FW			:BOOL;		//手动正转
	bJog_BW			:BOOL;	 //手动反转
	
	bRun_FW			:BOOL;		//正转
	bRun_BW			:BOOL;	 //反转
	
	bo_Pul			:BOOL;		//电机启动
	bo_Dir			:BOOL;//电机方向(0=正转)

END_STRUCT
END_TYPE

// ---- P2DUTs/01_AxisCO_Ntrol/ST_ECYCtrl.TcDUT
TYPE ST_ECYCtrl :
STRUCT
    bServON   :BOOL;   
    bHome      :BOOL;   
    bReset      :BOOL;   
    bStop         :BOOL;   
   bJog_P         :BOOL;   
   bJog_N        :BOOL;   
   Pos_Start      :BOOL;   
   fTagetPos     :REAL;
   fVel:           REAL;
   fAcc        :REAL;  
   fDec        :REAL;  
  // Delay_Time  :TIME;


